        // timeout exceeded ? 
        IF (CheckTimeout(_timerCmd) = RobotLibraryConstants.OK)
        THEN
          ErrorID     := RobotLibraryEvents.ERR_TIMEOUT_CMD;
          ErrorAddTxt := CONCAT('_stepCmd = ' , DINT_TO_STRING(_stepCmd));
        END_IF
      END_IF
  
  
  05: IF (( NOT ExchangeConfiguration.Busy              ) AND
          (     ExchangeConfiguration.ParameterAccepted ))
      THEN
        // stop execution       
        ExchangeConfiguration.Enable := FALSE;
        // set timeout
        SetTimeout(PT := _timeoutCmd, rTimer := _timerCmd);
        // inc step counter
       _stepCmd := _stepCmd + 1;       
       ELSE
         // check error ? 
         IF (ExchangeConfiguration.Error)
         THEN
           ErrorID     := ExchangeConfiguration.ErrorID;
           ErrorAddTxt := ExchangeConfiguration.ErrorAddTxt;;
         END_IF  
       
         // timeout exceeded ? 
         IF (CheckTimeout(_timerCmd) = RobotLibraryConstants.OK)
         THEN
           ErrorID     := RobotLibraryEvents.ERR_TIMEOUT_CMD;
           ErrorAddTxt := CONCAT('_stepCmd = ' , DINT_TO_STRING(_stepCmd));
         END_IF
       END_IF

       
  06: IF (( NOT ReadRobotData.Busy  ) AND 
          ( NOT ReadRobotData.Error )) 
      THEN
        // start function block
        ReadRobotData.Execute := TRUE;
        // set timeout
        SetTimeout(PT := _timeoutCmd, rTimer := _timerCmd);
        // inc step counter
       _stepCmd := _stepCmd + 1;       
      ELSE
        // check error ? 
        IF (ReadRobotData.Error)
        THEN
          ErrorID     := ReadRobotData.ErrorID;
          ErrorAddTxt := ReadRobotData.ErrorAddTxt;;
        END_IF  
        // timeout exceeded ? 
        IF (CheckTimeout(_timerCmd) = RobotLibraryConstants.OK)
        THEN
          ErrorID     := RobotLibraryEvents.ERR_TIMEOUT_CMD;
          ErrorAddTxt := CONCAT('_stepCmd = ' , DINT_TO_STRING(_stepCmd));
        END_IF
      END_IF
  
  07: IF ( ReadRobotData.Busy ) 
      THEN
        // set timeout
        SetTimeout(PT := _timeoutCmd, rTimer := _timerCmd);
        // inc step counter
       _stepCmd := _stepCmd + 1;       
      ELSE
        // check error ? 
        IF (ReadRobotData.Error)
        THEN
          ErrorID     := ReadRobotData.ErrorID;
          ErrorAddTxt := ReadRobotData.ErrorAddTxt;;
        END_IF  
       
        // timeout exceeded ? 
        IF (CheckTimeout(_timerCmd) = RobotLibraryConstants.OK)
        THEN
          ErrorID     := RobotLibraryEvents.ERR_TIMEOUT_CMD;
          ErrorAddTxt := CONCAT('_stepCmd = ' , DINT_TO_STRING(_stepCmd));
        END_IF
      END_IF
  
  
  08: IF (( NOT ReadRobotData.Busy  ) AND
          (     ReadRobotData.Done  ))
      THEN       
        // start function block
        ReadRobotData.Execute := FALSE;
        // set timeout
        SetTimeout(PT := _timeoutCmd, rTimer := _timerCmd);
        // inc step counter
       _stepCmd := _stepCmd + 1;
       ELSE
         // check error ? 
         IF (ReadRobotData.Error)
         THEN
           ErrorID     := ReadRobotData.ErrorID;
           ErrorAddTxt := ReadRobotData.ErrorAddTxt;;
         END_IF  
       
         // timeout exceeded ? 
         IF (CheckTimeout(_timerCmd) = RobotLibraryConstants.OK)
         THEN
           ErrorID     := RobotLibraryEvents.ERR_TIMEOUT_CMD;
           ErrorAddTxt := CONCAT('_stepCmd = ' , DINT_TO_STRING(_stepCmd));
         END_IF
       END_IF


  09: IF (( NOT ReadMessages.Busy  ) AND 
          ( NOT ReadMessages.Error )) 
      THEN
        // start function block
        ReadMessages.Enable := TRUE;
        // set timeout
        SetTimeout(PT := _timeoutCmd, rTimer := _timerCmd);
        // inc step counter
       _stepCmd := _stepCmd + 1;       
      ELSE
        // check error ? 
        IF (ReadMessages.Error)
        THEN
          ErrorID     := ReadMessages.ErrorID;
          ErrorAddTxt := ReadMessages.ErrorAddTxt;;
        END_IF  
        // timeout exceeded ? 
        IF (CheckTimeout(_timerCmd) = RobotLibraryConstants.OK)
        THEN
          ErrorID     := RobotLibraryEvents.ERR_TIMEOUT_CMD;
          ErrorAddTxt := CONCAT('_stepCmd = ' , DINT_TO_STRING(_stepCmd));
        END_IF
      END_IF
  
  10: IF ( ReadMessages.Busy )
      THEN
        // set timeout
        SetTimeout(PT := _timeoutCmd, rTimer := _timerCmd);
        // inc step counter
       _stepCmd := _stepCmd + 1;       
      ELSE
        // check error ? 
        IF (ReadMessages.Error)
        THEN
          ErrorID     := ReadMessages.ErrorID;
          ErrorAddTxt := ReadMessages.ErrorAddTxt;;
        END_IF  
       
        // timeout exceeded ? 
        IF (CheckTimeout(_timerCmd) = RobotLibraryConstants.OK)
        THEN
          ErrorID     := RobotLibraryEvents.ERR_TIMEOUT_CMD;
          ErrorAddTxt := CONCAT('_stepCmd = ' , DINT_TO_STRING(_stepCmd));
        END_IF
      END_IF
  
  
  11: IF ((     ReadMessages.Enabled ) AND
          ( NOT ReadMessages.Error   ))
      THEN       
        // set timeout
        SetTimeout(PT := _timeoutCmd, rTimer := _timerCmd);
        // inc step counter
       _stepCmd := _stepCmd + 1;
      ELSE
         // check error ? 
         IF (ReadRobotData.Error)
         THEN
           ErrorID     := ReadMessages.ErrorID;
           ErrorAddTxt := ReadMessages.ErrorAddTxt;;
         END_IF  
       
         // timeout exceeded ? 
         IF (CheckTimeout(_timerCmd) = RobotLibraryConstants.OK)
         THEN
           ErrorID     := RobotLibraryEvents.ERR_TIMEOUT_CMD;
           ErrorAddTxt := CONCAT('_stepCmd = ' , DINT_TO_STRING(_stepCmd));
         END_IF
       END_IF

  12:  // Reset busy flag
       Busy := FALSE;
       // set initialized flag
       Initialized := TRUE;
       
       // Wait for task disable
       IF ( NOT Enable)
       THEN
         // reset start of function blocks
         ReadMessages.Enable := FALSE;
         ReadRobotData.Execute := FALSE;
         ExchangeConfiguration.Enable := FALSE;
         // Reset step counter
        _stepCmd := 0;         
         // finished okay
         OnExecRun := RobotLibraryConstants.OK;
       END_IF  

       
ELSE
  // invalid step
  ErrorID     := RobotLibraryEvents.ERR_INVALID_STEP;
  ErrorAddTxt := CONCAT('_stepCmd = ' , DINT_TO_STRING(_stepCmd));
END_CASE


// Reset FB
IF ( OnExecRun <> RobotLibraryConstants.RUNNING)
THEN
 _stepCmd     := 0;
  Busy        := FALSE;
  Error       := FALSE;
  ErrorID     := 0;
  ErrorAddTxt := '';
  WarningID   := 0;
  InfoID      := 0;  
END_IF
END_METHOD

METHOD PRIVATE ParseRecvPayload
VAR_IN_OUT
  /// Robot assignment of function
  AxesGroup    : AxesGroup;
  /// Inputs of PLC for communication from RC
  RobotInData  : ARRAY[0..RobotLibraryParameter.ROBOT_IN_DATA_MAX ] OF BYTE;
END_VAR

VAR
  /// internal index
 _idx             : DINT;
  /// temporary DWORD
 _tmpDword        : DWORD;
  /// length of data block
 _dataBlockLength : UINT;
  /// internal payload length
 _payLoadLen      : DWORD;  
  /// internal payload pointer
 _payLoadPtr      : DWORD;  
  /// sequence counter
 _seqCount        : DINT;
END_VAR
// Reset payload
RecvData.Reset();
// Copy inputs to payload  
SysDepMemCpy( pDest := ADR(RecvData.Payload) , pSrc  := ADR(RobotInData), DataLen := RobotLibraryParameter.TELEGRAM_PAYLOAD_MAX +1);

// check new data to receive ? 
IF ( Telegram.RobToPlc.Sequence[0].Header.SEQ_ACK <> AxesGroup.InternalData.LastACK[0]) {warning 'ToDo: handle 2nd sequence'} 
THEN
  // delete old telegram data 
  SysDepMemSet(pDest := ADR(Telegram.RobToPlc), Value := 0 , DataLen := SIZEOF(Telegram.RobToPlc));
END_IF


ParseRecvPayloadHeader        ( AxesGroup := AxesGroup);
ParseRecvPayloadCyclic        ( AxesGroup := AxesGroup);
ParseRecvPayloadCyclicOptional( AxesGroup := AxesGroup);
ParseRecvPayloadSequence      ( AxesGroup := AxesGroup);
ParseRecvPayloadFooter        ( AxesGroup := AxesGroup);
ParseRecvPayloadLogging       ( AxesGroup := AxesGroup);


AxesGroup.InternalData.LastACK[0] := Telegram.RobToPlc.Sequence[0].Header.SEQ_ACK; 
AxesGroup.InternalData.LastACK[1] := Telegram.RobToPlc.Sequence[1].Header.SEQ_ACK;
END_METHOD

METHOD PRIVATE ParseRecvPayloadCyclic
VAR_IN_OUT
  /// Robot assignment of function
  AxesGroup: AxesGroup;
END_VAR
END_METHOD

METHOD PRIVATE ParseRecvPayloadCyclicOptional
VAR_IN_OUT
  /// Robot assignment of function
  AxesGroup    : AxesGroup;
END_VAR

VAR 
  /// internal index for loops
 _idx : DINT;
END_VAR
// AxesGroup.OptionalCyclic.RobToPlc.SubProgramData {{{
IF ( AxesGroup.CyclicOptional.RobToPlc.SubProgramData.Active )
THEN
  FOR _idx := 0 TO 25 {warning 'Add contant for DataMax'}
  DO
    Telegram.RobToPlc.CyclicOptional.SubProgramData.Data[_idx] := RecvData.GetByte(); 
  END_FOR
END_IF
// }}}
  
// AxesGroup.OptionalCyclic.RobToPlc.CartesianPos {{{
IF ( AxesGroup.CyclicOptional.RobToPlc.CartesianPosition.Active )
THEN
  Telegram.RobToPlc.CyclicOptional.CartesianPosition.X                    := RecvData.GetReal();
  Telegram.RobToPlc.CyclicOptional.CartesianPosition.Y                    := RecvData.GetReal();
  Telegram.RobToPlc.CyclicOptional.CartesianPosition.Z                    := RecvData.GetReal();
  Telegram.RobToPlc.CyclicOptional.CartesianPosition.Rx                   := RecvData.GetReal();
  Telegram.RobToPlc.CyclicOptional.CartesianPosition.Ry                   := RecvData.GetReal();
  Telegram.RobToPlc.CyclicOptional.CartesianPosition.Rz                   := RecvData.GetReal();
  Telegram.RobToPlc.CyclicOptional.CartesianPosition.Config               := RecvData.GetWord();
  Telegram.RobToPlc.CyclicOptional.CartesianPosition.Turns_J2_J1          := RecvData.GetByte();
  Telegram.RobToPlc.CyclicOptional.CartesianPosition.Turns_J4_J3          := RecvData.GetByte();
  Telegram.RobToPlc.CyclicOptional.CartesianPosition.Turns_J6_J5          := RecvData.GetByte();
  Telegram.RobToPlc.CyclicOptional.CartesianPosition.Turns_E1             := RecvData.GetByte();  
  Telegram.RobToPlc.CyclicOptional.CartesianPosition.E1                   := RecvData.GetReal();  
  Telegram.RobToPlc.CyclicOptional.CartesianPosition.ToolNo               := RecvData.GetUsint();
  Telegram.RobToPlc.CyclicOptional.CartesianPosition.FrameNo              := RecvData.GetUsint();
  Telegram.RobToPlc.CyclicOptional.CartesianPosition.CurrentlyUsedToolNo  := RecvData.GetUsint();
  Telegram.RobToPlc.CyclicOptional.CartesianPosition.CurrentlyUsedFrameNo := RecvData.GetUsint();
  Telegram.RobToPlc.CyclicOptional.CartesianPosition.Reserve_1            := RecvData.GetByte();
  Telegram.RobToPlc.CyclicOptional.CartesianPosition.Reserve_2            := RecvData.GetByte();  
END_IF
// }}}

// AxesGroup.OptionalCyclic.RobToPlc.JointPosition {{{
IF ( AxesGroup.CyclicOptional.RobToPlc.JointPosition.Active )
THEN
  Telegram.RobToPlc.CyclicOptional.JointPosition.J1         := RecvData.GetReal();
  Telegram.RobToPlc.CyclicOptional.JointPosition.J2         := RecvData.GetReal();
  Telegram.RobToPlc.CyclicOptional.JointPosition.J3         := RecvData.GetReal();
  Telegram.RobToPlc.CyclicOptional.JointPosition.J4         := RecvData.GetReal();
  Telegram.RobToPlc.CyclicOptional.JointPosition.J5         := RecvData.GetReal();
  Telegram.RobToPlc.CyclicOptional.JointPosition.J6         := RecvData.GetReal();
  Telegram.RobToPlc.CyclicOptional.JointPosition.E1         := RecvData.GetReal();
  Telegram.RobToPlc.CyclicOptional.JointPosition.E1_Reserve := RecvData.GetWord();
END_IF  
// }}}

// AxesGroup.OptionalCyclic.RobToPlc.CartesianForce {{{
IF ( AxesGroup.CyclicOptional.RobToPlc.Force.Active )
THEN
  Telegram.RobToPlc.CyclicOptional.Force.X  := RecvData.GetReal();
  Telegram.RobToPlc.CyclicOptional.Force.Y  := RecvData.GetReal();
  Telegram.RobToPlc.CyclicOptional.Force.Z  := RecvData.GetReal();
  Telegram.RobToPlc.CyclicOptional.Force.Rx := RecvData.GetReal();
  Telegram.RobToPlc.CyclicOptional.Force.Ry := RecvData.GetReal();
  Telegram.RobToPlc.CyclicOptional.Force.Rz := RecvData.GetReal();
END_IF  
// }}}    
  
// AxesGroup.OptionalCyclic.RobToPlc.Current {{{
IF ( AxesGroup.CyclicOptional.RobToPlc.Current.Active )
THEN
  Telegram.RobToPlc.CyclicOptional.Current.J1  := RecvData.GetReal();
  Telegram.RobToPlc.CyclicOptional.Current.J2  := RecvData.GetReal();
  Telegram.RobToPlc.CyclicOptional.Current.J3  := RecvData.GetReal();
  Telegram.RobToPlc.CyclicOptional.Current.J4  := RecvData.GetReal();
  Telegram.RobToPlc.CyclicOptional.Current.J5  := RecvData.GetReal();
  Telegram.RobToPlc.CyclicOptional.Current.J6  := RecvData.GetReal();
END_IF    
  
// AxesGroup.OptionalCyclic.RobToPlc.CartesianPosExt {{{
IF ( AxesGroup.CyclicOptional.RobToPlc.CartesianPositionExt.Active )
THEN
  Telegram.RobToPlc.CyclicOptional.CartesianPositionExt.E2 := RecvData.GetReal();
  Telegram.RobToPlc.CyclicOptional.CartesianPositionExt.E3 := RecvData.GetReal();
  Telegram.RobToPlc.CyclicOptional.CartesianPositionExt.E4 := RecvData.GetReal();
  Telegram.RobToPlc.CyclicOptional.CartesianPositionExt.E5 := RecvData.GetReal();
  Telegram.RobToPlc.CyclicOptional.CartesianPositionExt.E6 := RecvData.GetReal();
END_IF  
// }}}       
  
// AxesGroup.OptionalCyclic.RobToPlc.JointPosition {{{
IF ( AxesGroup.CyclicOptional.RobToPlc.JointPositionExt.Active )
THEN
  Telegram.RobToPlc.CyclicOptional.JointPositionExt.E2 := RecvData.GetReal();
  Telegram.RobToPlc.CyclicOptional.JointPositionExt.E3 := RecvData.GetReal();
  Telegram.RobToPlc.CyclicOptional.JointPositionExt.E4 := RecvData.GetReal();
  Telegram.RobToPlc.CyclicOptional.JointPositionExt.E5 := RecvData.GetReal();
  Telegram.RobToPlc.CyclicOptional.JointPositionExt.E6 := RecvData.GetReal();  
END_IF  
// }}}    
      
// AxesGroup.OptionalCyclic.RobToPlc.CartesianForceExt {{{
IF ( AxesGroup.CyclicOptional.RobToPlc.ForceExt.Active )
THEN
  Telegram.RobToPlc.CyclicOptional.ForceExt.E1  := RecvData.GetReal();
  Telegram.RobToPlc.CyclicOptional.ForceExt.E2  := RecvData.GetReal();
  Telegram.RobToPlc.CyclicOptional.ForceExt.E3  := RecvData.GetReal();
  Telegram.RobToPlc.CyclicOptional.ForceExt.E4  := RecvData.GetReal();
  Telegram.RobToPlc.CyclicOptional.ForceExt.E5  := RecvData.GetReal();
  Telegram.RobToPlc.CyclicOptional.ForceExt.E6  := RecvData.GetReal();
END_IF
// }}}    
  
// AxesGroup.OptionalCyclic.RobToPlc.CurrentExt {{{
IF ( AxesGroup.CyclicOptional.RobToPlc.CurrentExt.Active )
THEN
  Telegram.RobToPlc.CyclicOptional.CurrentExt.E1  := RecvData.GetReal();
  Telegram.RobToPlc.CyclicOptional.CurrentExt.E2  := RecvData.GetReal();
  Telegram.RobToPlc.CyclicOptional.CurrentExt.E3  := RecvData.GetReal();
  Telegram.RobToPlc.CyclicOptional.CurrentExt.E4  := RecvData.GetReal();
  Telegram.RobToPlc.CyclicOptional.CurrentExt.E5  := RecvData.GetReal();
  Telegram.RobToPlc.CyclicOptional.CurrentExt.E6  := RecvData.GetReal();
END_IF
// }}}
END_METHOD

METHOD PRIVATE ParseRecvPayloadFooter
VAR_IN_OUT
  /// Robot assignment of function
  AxesGroup : AxesGroup;
END_VAR

VAR
  /// index of lifesign in footer
  _lifeSignIdxFooter : DINT;
END_VAR
IF (( _parCfg.Com.TelegramLengthRobToPlc    >= 1                                          ) AND 
    ( _parCfg.Com.TelegramLengthRobToPlc -1 <= RobotLibraryParameter.TELEGRAM_PAYLOAD_MAX ))
THEN
  // set index of last byte
 _lifeSignIdxFooter := _parCfg.Com.TelegramLengthRobToPlc -1;
 

  Telegram.RobToPlc.Footer.LifeSign := GetHalfeByteHi(RecvData.Payload[_lifeSignIdxFooter]); 
END_IF
END_METHOD

METHOD PRIVATE ParseRecvPayloadHeader
VAR_IN_OUT
  /// Robot assignment of function
  AxesGroup    : AxesGroup;
END_VAR
// Version
Telegram.RobToPlc.Header.SRCIVersion := ByteToVersion(RecvData.GetByte());
// Connection alive signal
Telegram.RobToPlc.Header.LifeSign    := RecvData.GetHalfeByte2(IncPayloadPtr := TRUE);
// Reserved byte
Telegram.RobToPlc.Header.Reserved       := RecvData.GetByte();
// Initialization and Telegram control state
Telegram.RobToPlc.Header.TelegramState  := RecvData.GetUsint();
// Combination of various RA related states.
Telegram.RobToPlc.Header.StatusRobotArm := RecvData.GetDword();
// Actual override in percentage encoding 
Telegram.RobToPlc.Header.Override       := RecvData.GetUint();
END_METHOD

METHOD PRIVATE ParseRecvPayloadLogging
VAR_IN_OUT
  /// Robot assignment of function
  AxesGroup    : AxesGroup;
END_VAR

VAR
  /// internal sequence index for loops
  _seqIdx : DINT;
  /// internal fragment index for loops
  _fragIdx : DINT;
END_VAR
RETURN;
FOR _seqIdx := 0 TO AxesGroup.InternalData.SequenceCountRecv
DO
  // check new data to receive ? 
  IF ( Telegram.RobToPlc.Sequence[_seqIdx].Header.SEQ_ACK <> AxesGroup.InternalData.LastACK[_seqIdx]) 
  THEN
    // Check sequence payload > 0 ?    
    IF (Telegram.RobToPlc.Sequence[_seqIdx].Header.PayloadLength > 0)
    THEN
      // Create log entry
      CreateLogMessagePara4 ( Timestamp   := SystemTime,
                              MessageType := MessageType.CMD,
                              Severity    := Severity.DEBUG,
                              MessageCode := 0,
                              MessageText := 'RecvData: ACK = {1}, received Sequence [{2}] with PayloadLength = {3}, Lifesign = {4}',
                              Para1       :=  UINT_TO_STRING(Telegram.RobToPlc.Sequence[_seqIdx].Header.SEQ_ACK),
                              Para2       :=  DINT_TO_STRING(_seqIdx),
                              Para3       :=  UINT_TO_STRING(Telegram.RobToPlc.Sequence[_seqIdx].Header.PayloadLength),
                              Para4       :=  BYTE_TO_STRING(Telegram.RobToPlc.Header.LifeSign));
  
      FOR _fragIdx := 0 TO AxesGroup.InternalData.FragmentCountRecv[_seqIdx] 
      DO
        // Check fragment payload > 0 ?    
        IF (Telegram.RobToPlc.Sequence[_seqIdx].Fragment[_fragIdx].Header.PayloadLength > 0)
        THEN
          // Create log entry
          CreateLogMessagePara5 ( Timestamp   := SystemTime,
                                  MessageType := MessageType.CMD,
                                  Severity    := Severity.DEBUG,
                                  MessageCode := 0,
                                  MessageText := 'RecvData: received Fragment [{1}] with PayloadLength = {2}, CmdID <{3}> , CmdState: {4}, Fragment-Action Bits: {5}',
                                  Para1       :=  DINT_TO_STRING(0), {warning 'Add seqIdx'}
                                  Para2       :=  UINT_TO_STRING              (Telegram.RobToPlc.Sequence[_seqIdx].Fragment[_fragIdx].Header.PayloadLength),
                                  Para3       :=  DINT_TO_STRING              (Telegram.RobToPlc.Sequence[_seqIdx].Fragment[_fragIdx].Header.CmdID),
                                  Para4       :=  CMD_MESSAGE_STATE_TO_STRING (Telegram.RobToPlc.Sequence[_seqIdx].Fragment[_fragIdx].Command.Header.State),
                                  Para5       :=    FRAGMENT_ACTION_TO_STRING (Telegram.RobToPlc.Sequence[_seqIdx].Fragment[_fragIdx].Header.FragmentAction));
        END_IF
      END_FOR    
    END_IF
  END_IF
END_FOR
END_METHOD

METHOD PRIVATE ParseRecvPayloadSequence
VAR_IN_OUT
  /// Robot assignment of function
  AxesGroup    : AxesGroup;
END_VAR

VAR
  /// internal index
 _idx             : DINT;
  /// temporary DWORD
 _tmpDword        : DWORD;
  /// length of data block
 _dataBlockLength : UINT;
  /// internal payload length
 _payLoadLen      : DWORD;  
  /// internal payload pointer
 _payLoadPtr      : DWORD;  
  /// sequence counter
 _seqCount        : DINT;
END_VAR


VAR_INST
  /// last received acknowledge
 _lastACK : ARRAY[0..1] OF UDINT;
END_VAR
// Sequence Data
Telegram.RobToPlc.Sequence[0].Header.SEQ_ACK       := RecvData.GetUint();
Telegram.RobToPlc.Sequence[0].Header.PayloadLength := RecvData.GetUint();

// check new data ? 
IF ( Telegram.RobToPlc.Sequence[0].Header.SEQ_ACK <> AxesGroup.InternalData.LastACK[0]) {warning 'ToDo Handle 2nd sequence'} 
THEN

  IF (Telegram.RobToPlc.Sequence[0].Header.PayloadLength > 0)
  THEN
    // Create log entry
    CreateLogMessagePara4 ( Timestamp   := SystemTime,
                            MessageType := MessageType.CMD,
                            Severity    := Severity.DEBUG,
                            MessageCode := 0,
                            MessageText := 'RecvData: ACK = {1}, received Sequence [{2}] with PayloadLength = {3}, Lifesign = {4}',
                            Para1       :=  UINT_TO_STRING(Telegram.RobToPlc.Sequence[0].Header.SEQ_ACK),
                            Para2       :=  DINT_TO_STRING(0), {warning 'Add seqIdx'}
                            Para3       :=  UINT_TO_STRING(Telegram.RobToPlc.Sequence[0].Header.PayloadLength),
                            Para4       :=  BYTE_TO_STRING(Telegram.RobToPlc.Header.LifeSign));
    
    Telegram.RobToPlc.Sequence[0].Fragment[0].Header.CmdID               := RecvData.GetUint();
    Telegram.RobToPlc.Sequence[0].Fragment[0].Header.Reserve             := RecvData.GetByte();
    Telegram.RobToPlc.Sequence[0].Fragment[0].Header.FragmentAction      := RecvData.GetByte();
    Telegram.RobToPlc.Sequence[0].Fragment[0].Header.PayloadPointer      := RecvData.GetUint();
    Telegram.RobToPlc.Sequence[0].Fragment[0].Header.PayloadLength       := RecvData.GetUint();
    
    
    IF (Telegram.RobToPlc.Sequence[0].Fragment[0].Header.PayloadLength > 0)
    THEN
      // Fill Respone payload
      FOR _idx := Telegram.RobToPlc.Sequence[0].Fragment[0].Header.PayloadPointer TO Telegram.RobToPlc.Sequence[0].Fragment[0].Header.PayloadLength
      DO
        Telegram.RobToPlc.Sequence[0].Fragment[0].Command.Payload[_idx] := RecvData.GetByte();
      END_FOR
      
      // Add Response to ACR
      AxesGroup.Acyclic.ActiveCommandRegister.AddRsp(Telegram.RobToPlc.Sequence[0].Fragment[0]);
    
      // Only for debugging
      Telegram.RobToPlc.Sequence[0].Fragment[0].Command.Header.State                 := GetHalfeByteLo(Telegram.RobToPlc.Sequence[0].Fragment[0].Command.Payload[0]);
      Telegram.RobToPlc.Sequence[0].Fragment[0].Command.Header.ParSeq                := GetHalfeByteHi(Telegram.RobToPlc.Sequence[0].Fragment[0].Command.Payload[0]);
      Telegram.RobToPlc.Sequence[0].Fragment[0].Command.Header.AlarmMessageSeverity  :=   BYTE_TO_SINT(Telegram.RobToPlc.Sequence[0].Fragment[0].Command.Payload[1]);
      Telegram.RobToPlc.Sequence[0].Fragment[0].Command.Header.AlarmMessageCode      :=  CombineBytesToUint( HiByte := Telegram.RobToPlc.Sequence[0].Fragment[0].Command.Payload[2],
                                                                                                             LoByte := Telegram.RobToPlc.Sequence[0].Fragment[0].Command.Payload[3]);
      // Create log entry
      CreateLogMessagePara5 ( Timestamp   := SystemTime,
                              MessageType := MessageType.CMD,
                              Severity    := Severity.DEBUG,
                              MessageCode := 0,
                              MessageText := 'RecvData: received Fragment [{1}] with PayloadLength = {2}, CmdID <{3}> , CmdState: {4}, Fragment-Action Bits: {5}',
                              Para1       :=  DINT_TO_STRING(0), {warning 'Add seqIdx'}
                              Para2       :=  UINT_TO_STRING              (Telegram.RobToPlc.Sequence[0].Fragment[0].Header.PayloadLength),
                              Para3       :=  DINT_TO_STRING              (Telegram.RobToPlc.Sequence[0].Fragment[0].Header.CmdID),
                              Para4       :=  CMD_MESSAGE_STATE_TO_STRING (Telegram.RobToPlc.Sequence[0].Fragment[0].Command.Header.State),
                              Para5       :=    FRAGMENT_ACTION_TO_STRING (Telegram.RobToPlc.Sequence[0].Fragment[0].Header.FragmentAction));
                              //Para6       :=  BYTE_TO_STRING(Telegram.RobToPlc.Header.LifeSign)
    END_IF    
  END_IF
END_IF  

IF ( RobotLibraryParameter.TWO_SEQUENCES ) {warning 'ToDo'}
THEN
 _seqCount := _seqCount + 1;
END_IF
END_METHOD

END_FUNCTION_BLOCK

// Library/POUs/Read/MC_ReadRobotData/MC_ReadRobotDataFB
/// Read robot-specific data from the RC
FUNCTION_BLOCK MC_ReadRobotDataFB EXTENDS RobotLibraryBaseExecuteFB
// ------------------------------------------------------------------------- 
//  SRCI Robot Library                                                
// ------------------------------------------------------------------------- 
//                                                                           
//  Object:      ReadRobotDataFB                                       
//  Author:      Thorsten Brach                                                
//  Date:        2024-08-11
//
//  Description:                                              
//   
//                                                                           
//  Copyright: 
//    (C) 2024 Thorsten Brach. All rights reserved                                                                                                                                            
//             Licensed under the LGPL-3.0 license.
//                                                                           
//  Disclaimer:                                                                           
//    This project is provided without any guarantee and can be used for   
//    private and commercial purposes. Any use is at the user’s 
//    own risk and responsibility.
//
// -------------------------------------------------------------------------
VAR_INPUT
  /// internal copy of command parameter 
  ParCmd          : ReadRobotDataParCmd;  
END_VAR

VAR_OUTPUT
  /// Command is transferred and confirmed by the RC
  CommandBuffered : BOOL;
  /// command outputs
  OutCmd          : ReadRobotDataOutCmd;       
END_VAR


VAR
  /// internal copy of command parameter 
 _parCmd             : ReadRobotDataParCmd;
  /// command data to send
 _command            : ReadRobotDataSendData;
  /// response data received
 _response           : ReadRobotDataRecvData;      
END_VAR

SUPER^(AxesGroup := AxesGroup);

METHOD PROTECTED CheckFunctionSupported : BOOL
VAR_IN_OUT
  /// Robot assignment of function
  AxesGroup : AxesGroup; 
END_VAR
CheckFunctionSupported := AxesGroup.InternalData.RCSupportedFunctions.ReadRobotData;

IF ( NOT CheckFunctionSupported )
THEN
  // call base implementation for set error and create log entry
  SUPER^.CheckFunctionSupported(AxesGroup := AxesGroup);
END_IF
END_METHOD

METHOD PROTECTED CheckParameterChanged : BOOL
VAR_IN_OUT
  /// Robot assignment of function
  AxesGroup    : AxesGroup; 
END_VAR
// Check ParCmd Size is > 0, because MemCmp does not work correctly with size = 0
IF (SIZEOF(ParCmd) = 0) 
THEN 
  RETURN;
END_IF

// compare memory 
_parameterChanged := ( SysDepMemCmp(pData1 := ADR(ParCmd), pData2 := ADR(_parCmd), DataLen := SIZEOF(ParCmd)) <> RobotLibraryConstants.OK );

// check parameter valid ?
_parameterValid   := CheckParameterValid( AxesGroup := AxesGroup );

IF ((  _parameterChanged        )  AND 
    (  _parameterValid          )) OR
    (  _parameterUpdateInternal )  
THEN  
  // reset internal flag for send parameter update
 _parameterUpdateInternal := FALSE;
  // update internal copy of parameters 
 _parCmd := ParCmd;
  // inc parameter sequence
 _command.ParSeq := _command.ParSeq + 1;
  // update command data  
  CommandData := CreateCommandPayload(AxesGroup := AxesGroup); // ( Access via reference to rCommandFB in ACR )
  // notify active command register 
  AxesGroup.Acyclic.ActiveCommandRegister.NotifyParameterChanged := _uniqueID;
END_IF
END_METHOD

METHOD INTERNAL CreateCommandPayload : RobotLibrarySendDataFB
VAR_IN_OUT
  /// Robot assignment of function
  AxesGroup : AxesGroup; 
END_VAR
// Table 6-17: Sent CMD payload (PLC to RC) of "ReadRobotData"
// --------------------------
// Header
// --------------------------
// Byte 00 : UINT  - Type HB     
// Byte 01 :       - Type LB    
// Byte 02 : USINT - Reserve | ExecutionMode
// Byte 03 : USINT - ParSeq  | Priority
// --------------------------
// set command parameter 
_command.CmdTyp   :=  CmdType.ReadRobotData;
_command.ExecMode :=  ExecMode;
_command.ParSeq   := _command.ParSeq;
_command.Priority :=  Priority;

// copy command data to header
_cmdHeader := _command;
// call base implementation to copy header to payload buffer
CreateCommandPayload := SUPER^.CreateCommandPayload(AxesGroup := AxesGroup);

// Create logging
CreateCommandPayloadLog(AxesGroup := AxesGroup);
END_METHOD

METHOD INTERNAL CreateCommandPayloadLog
VAR_IN_OUT
  /// Robot assignment of function
  AxesGroup : AxesGroup; 
END_VAR
// Create log entry for Parameter start
CreateLogMessage      ( Timestamp   := AxesGroup.InternalData.SystemTime,
                        MessageType := MessageType.CMD,
                        Severity    := Severity.DEBUG,
                        MessageCode := 0,
                        MessageText := 'Create command payload without additional parameter(s)');
END_METHOD

METHOD FB_init : BOOL
VAR_INPUT
  /// if TRUE, the retain variables are initialized (warm start / cold start)
  bInitRetains : BOOL; 
  /// if TRUE, the instance afterwards gets moved into the copy code (online change)
  bInCopyCode  : BOOL;  
END_VAR
MyType := 'MC_ReadRobotDataFB';
ExecMode := ExecutionMode.PARALLEL;
END_METHOD

METHOD PROTECTED OnCall
VAR_IN_OUT
  /// Robot assignment of function
  AxesGroup : AxesGroup; 
END_VAR
// call base implementation
SUPER^.OnCall(AxesGroup := AxesGroup);

CASE _stepCmd OF
  
  00:  IF ( _execute_R.Q )  
       THEN
         // Check function is supported and parameter are valid ?
         IF (( CheckFunctionSupported( AxesGroup := AxesGroup )) AND
             ( CheckParameterValid   ( AxesGroup := AxesGroup )))
         THEN      
           // set busy flag
           Busy := TRUE;
           // Reset command outputs
           SysDepMemSet(pDest := ADR(OutCmd), Value := 0, DataLen := SIZEOF(OutCmd));         
           // apply command parameter
          _parCmd := ParCmd;
           // init parameter sequence
          _command.ParSeq := 1;
           // create command data
           CommandData := CreateCommandPayload(AxesGroup := AxesGroup);
           // Add command to active command register
          _uniqueID := AxesGroup.Acyclic.ActiveCommandRegister.AddCmd( pCommandFB := ADR(THIS^ ));     
           // set timeout
           SetTimeout(PT := _timeoutCmd, rTimer := _timerCmd);
           // inc step counter
          _stepCmd := _stepCmd + 1; 
         END_IF
       END_IF
     

  01:  // Wait for responce received
       IF ( _responseReceived )
       THEN
         // reset response received flag
        _responseReceived := FALSE;

         CASE  _response.State 
         OF
           CmdMessageState.BUFFERED    : CommandBuffered    := TRUE;
           CmdMessageState.DONE        : Done               := TRUE;
           CmdMessageState.ERROR       : Error              := TRUE;
         END_CASE
                
         // Done, Aborted or Error ?
         IF (_response.State >= CmdMessageState.DONE )
         THEN
           // reset Busy Flag
           Busy := FALSE;
           // Update results
           OutCmd.RCManufacturer       :=                              _response.RCManufacturer;
           OutCmd.RCOrderID            :=                              _response.RCOrderID;
           OutCmd.RCSerialNumber       :=                              _response.RCSerialNumber;
           OutCmd.RASerialNumber       :=                              _response.RASerialNumber;
           OutCmd.RCFirmwareVersion    :=                              _response.RCFirmwareVersion;
           OutCmd.RCInterpreterVersion :=                              _response.RCInterpreterVersion;
           OutCmd.AxisJointUsed        :=                              _response.AxisJointUsed;
           OutCmd.AxisExternalUsed     :=                              _response.AxisExternalUsed;
           OutCmd.AxisJointUnit        :=                              _response.AxisJointUnit;
           OutCmd.AxisExternalUnit     :=                              _response.AxisExternalUnit;
           OutCmd.RCSupportedFunctions :=  BytesToRCSupportedFunctions(_response.RCSupportedFunctions);
           OutCmd.RobotID              :=                              _response.RobotID;  
           OutCmd.InterpreterCycleTime :=                              _response.InterpreterCycleTime;
           // set timeout
           SetTimeout(PT := _timeoutCmd, rTimer := _timerCmd);
           // inc step counter
          _stepCmd := _stepCmd + 1; 
         END_IF
       END_IF


  02: IF ( NOT Execute)
      THEN
        Reset();
      END_IF     

ELSE
  // invalid step
  ErrorID := RobotLibraryEvents.ERR_INVALID_STEP;
END_CASE


// Reset FB
IF ( NOT Execute )
THEN
  Reset(); 
END_IF
END_METHOD

METHOD INTERNAL ParseResponsePayload : DINT
VAR_INPUT
  /// Response data
  ResponseData : RobotLibraryRecvDataFB;
  /// Timestamp
  Timestamp    : SystemTime;  
END_VAR
// Table 6-18: Received CMD payload (RC to PLC) of "ReadRobotData"
// --------------------------
// Header
// --------------------------
// Byte 00 : USINT   - ParSeq | State     
// Byte 01 : SINT    - AlarmMessageSeverity    
// Byte 02 : UINT    - AlarmMessageCode HB
// Byte 03 :         - AlarmMessageCode LB
// --------------------------
// Datablock
// --------------------------
// Byte 04 : CHAR  RCManufacturer[0];
// Byte 05 : CHAR  RCManufacturer[1];
// Byte 06 : CHAR  RCManufacturer[2];
// Byte 07 : CHAR  RCManufacturer[3];
// Byte 08 : CHAR  RCManufacturer[4];
// Byte 09 : CHAR  RCManufacturer[5];
// Byte 10 : CHAR  RCManufacturer[6];
// Byte 11 : CHAR  RCManufacturer[7];
// Byte 12 : CHAR  RCManufacturer[8];
// Byte 13 : CHAR  RCManufacturer[9];
// Byte 14 : CHAR  RCManufacturer[10];
// Byte 15 : CHAR  RCManufacturer[11];
// Byte 16 : CHAR  RCManufacturer[12];
// Byte 17 : CHAR  RCManufacturer[13];
// Byte 18 : CHAR  RCManufacturer[14];
// Byte 19 : CHAR  RCManufacturer[15];
// Byte 20 : CHAR  RCManufacturer[16];
// Byte 21 : CHAR  RCManufacturer[17];
// Byte 22 : CHAR  RCManufacturer[18];
// Byte 23 : CHAR  RCManufacturer[19];
// Byte 24 : CHAR  RCOrderID[0];
// Byte 25 : CHAR  RCOrderID[1];
// Byte 26 : CHAR  RCOrderID[2];
// Byte 27 : CHAR  RCOrderID[3];
// Byte 28 : CHAR  RCOrderID[4];
// Byte 29 : CHAR  RCOrderID[5];
// Byte 30 : CHAR  RCOrderID[6];
// Byte 31 : CHAR  RCOrderID[7];
// Byte 32 : CHAR  RCOrderID[8];
// Byte 33 : CHAR  RCOrderID[9];
// Byte 34 : CHAR  RCOrderID[10];
// Byte 35 : CHAR  RCOrderID[11];
// Byte 36 : CHAR  RCOrderID[12];
// Byte 37 : CHAR  RCOrderID[13];
// Byte 38 : CHAR  RCOrderID[14];
// Byte 39 : CHAR  RCOrderID[15];
// Byte 40 : CHAR  RCOrderID[16];
// Byte 41 : CHAR  RCOrderID[17];
// Byte 42 : CHAR  RCOrderID[18];
// Byte 43 : CHAR  RCOrderID[19];
// Byte 44 : CHAR  RCSerialNumber[0];
// Byte 45 : CHAR  RCSerialNumber[1];
// Byte 46 : CHAR  RCSerialNumber[2];
// Byte 47 : CHAR  RCSerialNumber[3];
// Byte 48 : CHAR  RCSerialNumber[4];
// Byte 49 : CHAR  RCSerialNumber[5];
// Byte 50 : CHAR  RCSerialNumber[6];
// Byte 51 : CHAR  RCSerialNumber[7];
// Byte 52 : CHAR  RCSerialNumber[8];
// Byte 53 : CHAR  RCSerialNumber[9];
// Byte 54 : CHAR  RCSerialNumber[10];
// Byte 55 : CHAR  RCSerialNumber[11];
// Byte 56 : CHAR  RCSerialNumber[12];
// Byte 57 : CHAR  RCSerialNumber[13];
// Byte 58 : CHAR  RCSerialNumber[14];
// Byte 59 : CHAR  RCSerialNumber[15];
// Byte 60 : CHAR  RASerialNumber[0];
// Byte 61 : CHAR  RASerialNumber[1];
// Byte 62 : CHAR  RASerialNumber[2];
// Byte 63 : CHAR  RASerialNumber[3];
// Byte 64 : CHAR  RASerialNumber[4];
// Byte 65 : CHAR  RASerialNumber[5];
// Byte 66 : CHAR  RASerialNumber[6];
// Byte 67 : CHAR  RASerialNumber[7];
// Byte 68 : CHAR  RASerialNumber[8];
// Byte 69 : CHAR  RASerialNumber[9];
// Byte 70 : CHAR  RASerialNumber[10];
// Byte 71 : CHAR  RASerialNumber[11];
// Byte 72 : CHAR  RASerialNumber[12];
// Byte 73 : CHAR  RASerialNumber[13];
// Byte 74 : CHAR  RASerialNumber[14];
// Byte 75 : CHAR  RASerialNumber[15];
// Byte 76 : CHAR  RCFirmwareVersion[0];
// Byte 77 : CHAR  RCFirmwareVersion[1];
// Byte 78 : CHAR  RCFirmwareVersion[2];
// Byte 79 : CHAR  RCFirmwareVersion[3];
// Byte 80 : CHAR  RCFirmwareVersion[4];
// Byte 81 : CHAR  RCFirmwareVersion[5];
// Byte 82 : CHAR  RCFirmwareVersion[6];
// Byte 83 : CHAR  RCFirmwareVersion[7];
// Byte 84 : CHAR  RCFirmwareVersion[8];
// Byte 85 : CHAR  RCFirmwareVersion[9];
// Byte 86 : CHAR  RCFirmwareVersion[10];
// Byte 87 : CHAR  RCFirmwareVersion[11];
// Byte 88 : CHAR  RCInterpreterVersion[0];
// Byte 89 : CHAR  RCInterpreterVersion[1];
// Byte 90 : CHAR  RCInterpreterVersion[2];
// Byte 91 : BYTE  Reserved;
// Byte 92 : BYTE  AxisJointUsed;
// Byte 93 : BYTE  AxisExternalUsed;
// Byte 94 : BYTE  AxisJointUnit;
// Byte 95 : BYTE  AxisExternalUnit;
// Byte 96 : BYTE  RCSupportedFunctions[0];
// Byte 97 : BYTE  RCSupportedFunctions[1];
// Byte 98 : BYTE  RCSupportedFunctions[2];
// Byte 99 : BYTE  RCSupportedFunctions[3];
// Byte 100: BYTE  RCSupportedFunctions[4];
// Byte 101: BYTE  RCSupportedFunctions[5];
// Byte 102: BYTE  RCSupportedFunctions[6];
// Byte 103: BYTE  RCSupportedFunctions[7];
// Byte 104: BYTE  RCSupportedFunctions[8];
// Byte 105: BYTE  RCSupportedFunctions[9];
// Byte 106: BYTE  RCSupportedFunctions[10];
// Byte 107: BYTE  RCSupportedFunctions[11];
// Byte 108: BYTE  RCSupportedFunctions[12];
// Byte 109: BYTE  RCSupportedFunctions[13];
// Byte 110: BYTE  RCSupportedFunctions[14];
// Byte 111: BYTE  RCSupportedFunctions[15];
// Byte 112: BYTE  RCSupportedFunctions[16];
// Byte 113: BYTE  RCSupportedFunctions[17];
// Byte 114: BYTE  RCSupportedFunctions[18];
// Byte 115: BYTE  Reserved;
// Byte 116: CHAR  RobotID[0];
// Byte 117: CHAR  RobotID[1];
// Byte 118: CHAR  RobotID[2];
// Byte 119: CHAR  RobotID[3];
// Byte 120: CHAR  RobotID[4];
// Byte 121: CHAR  RobotID[5];
// Byte 122: CHAR  RobotID[6];
// Byte 123: CHAR  RobotID[7];
// Byte 124: CHAR  RobotID[8];
// Byte 125: CHAR  RobotID[9];
// Byte 126: CHAR  RobotID[10];
// Byte 127: CHAR  RobotID[11];
// Byte 128: CHAR  RobotID[12];
// Byte 129: CHAR  RobotID[13];
// Byte 130: CHAR  RobotID[14];
// Byte 131: CHAR  RobotID[15];
// Byte 132: UINT  InterpreterCycleTime HW HB;
// Byte 133:       InterpreterCycleTime HW LB;
// --------------------------
// call base implementation to parse the header from payload buffer
ResponseData.PayloadPtr := SUPER^.ParseResponsePayload(ResponseData := ResponseData, Timestamp := Timestamp);

// copy parsed header to response
_response.ParSeq               := _rspHeader.ParSeq;
_response.State                := _rspHeader.State;
_response.AlarmMessageSeverity := _rspHeader.AlarmMessageSeverity;
_response.AlarmMessageCode     := _rspHeader.AlarmMessageCode;

// Get _response.RCManufacturer
ResponseData.GetDataBlock(pData := ADR(_response.RCManufacturer)      , SIZEOF(_response.RCManufacturer   )   , IsString := TRUE );
// Get _response.RCOrderID
ResponseData.GetDataBlock(pData := ADR(_response.RCOrderID)           , SIZEOF(_response.RCOrderID        )   , IsString := TRUE );
// Get _response.RCSerialNumber
ResponseData.GetDataBlock(pData := ADR(_response.RCSerialNumber)      , SIZEOF(_response.RCSerialNumber   )   , IsString := TRUE );
// Get _response.RASerialNumber
ResponseData.GetDataBlock(pData := ADR(_response.RASerialNumber)      , SIZEOF(_response.RASerialNumber   )   , IsString := TRUE );
// Get _response.RCFirmwareVersion
ResponseData.GetDataBlock(pData := ADR(_response.RCFirmwareVersion)   , SIZEOF(_response.RCFirmwareVersion)   , IsString := TRUE );
// Get _response.RCInterpreterVersion
ResponseData.GetDataBlock(pData := ADR(_response.RCInterpreterVersion), SIZEOF(_response.RCInterpreterVersion), IsString := TRUE );

// Get _response.Reserve
_response.Reserve := ResponseData.GetByte(); 
// Get _response.AxisJointUsed
_response.AxisJointUsed := ResponseData.GetByte(); 
// Get _response.AxisExternalUsed
_response.AxisExternalUsed := ResponseData.GetByte(); 
// Get _response.AxisJointUnit
_response.AxisJointUnit := ResponseData.GetByte(); 
// Get _response.AxisExternalUnit
_response.AxisExternalUnit := ResponseData.GetByte();
// Get _response.RCSupportedFunctions
ResponseData.GetDataBlock(pData := ADR(_response.RCSupportedFunctions), SIZEOF(_response.RCSupportedFunctions), IsString := FALSE );
// Get _response.Reserve2
_response.Reserve2 := ResponseData.GetByte(); 
// Get _response.RobotID
ResponseData.GetDataBlock(pData := ADR(_response.RobotID)             , SIZEOF(_response.RobotID)             , IsString := TRUE );
// Get _response.InterpreterCycleTime
_response.InterpreterCycleTime := ResponseData.GetUsint(); 

// Create logging
ParseResponsePayloadLog(ResponseData := ResponseData, Timestamp := Timestamp);
END_METHOD

METHOD INTERNAL ParseResponsePayloadLog
VAR_INPUT
  /// Response data
  ResponseData : RobotLibraryRecvDataFB;
  /// Timestamp
  Timestamp    : SystemTime;  
END_VAR
VAR 
  /// internal index for loops
 _idx : DINT;
  /// temporary string
 _tmpStr : STRING;
END_VAR
// Create log entry for Parameter start
CreateLogMessage      ( Timestamp   := Timestamp,
                        MessageType := MessageType.CMD,
                        Severity    := Severity.DEBUG,
                        MessageCode := 0,
                        MessageText := 'Parsed the following parameter(s) from response data:');

// Create log entry for RCManufacturer
CreateLogMessagePara1 ( Timestamp   := Timestamp,
                        MessageType := MessageType.CMD,
                        Severity    := Severity.DEBUG,
                        MessageCode := 0,
                        MessageText := 'Response.RCManufacturer = {1}',
                        Para1       := _response.RCManufacturer);

// Create log entry for RCOrderID
CreateLogMessagePara1 ( Timestamp   := Timestamp,
                        MessageType := MessageType.CMD,
                        Severity    := Severity.DEBUG,
                        MessageCode := 0,
                        MessageText := 'Response.RCOrderID = {1}',
                        Para1       := _response.RCOrderID);

// Create log entry for RCSerialNumber
CreateLogMessagePara1 ( Timestamp   := Timestamp,
                        MessageType := MessageType.CMD,
                        Severity    := Severity.DEBUG,
                        MessageCode := 0,
                        MessageText := 'Response.RCSerialNumber = {1}',
                        Para1       := _response.RCSerialNumber);

// Create log entry for RASerialNumber
CreateLogMessagePara1 ( Timestamp   := Timestamp,
                        MessageType := MessageType.CMD,
                        Severity    := Severity.DEBUG,
                        MessageCode := 0,
                        MessageText := 'Response.RASerialNumber = {1}',
                        Para1       := _response.RASerialNumber);

// Create log entry for RCFirmwareVersion
CreateLogMessagePara1 ( Timestamp   := Timestamp,
                        MessageType := MessageType.CMD,
                        Severity    := Severity.DEBUG,
                        MessageCode := 0,
                        MessageText := 'Response.RCFirmwareVersion = {1}',
                        Para1       := _response.RCFirmwareVersion);
                        
// Create log entry for RCInterpreterVersion
CreateLogMessagePara1 ( Timestamp   := Timestamp,
                        MessageType := MessageType.CMD,
                        Severity    := Severity.DEBUG,
                        MessageCode := 0,
                        MessageText := 'Response.RCInterpreterVersion = {1}',
                        Para1       := _response.RCInterpreterVersion);

// Create log entry for Reserve
CreateLogMessagePara1 ( Timestamp   := Timestamp,
                        MessageType := MessageType.CMD,
                        Severity    := Severity.DEBUG,
                        MessageCode := 0,
                        MessageText := 'Response.Reserve = {1}',
                        Para1       :=  BYTE_TO_STRING(_response.Reserve));

// Create log entry for AxisJointUsed
CreateLogMessagePara1 ( Timestamp   := Timestamp,
                        MessageType := MessageType.CMD,
                        Severity    := Severity.DEBUG,
                        MessageCode := 0,
                        MessageText := 'Response.AxisJointUsed = {1}',
                        Para1       :=  BYTE_TO_STRING_BIN(_response.AxisJointUsed));

// Create log entry for AxisExternalUsed
CreateLogMessagePara1 ( Timestamp   := Timestamp,
                        MessageType := MessageType.CMD,
                        Severity    := Severity.DEBUG,
                        MessageCode := 0,
                        MessageText := 'Response.AxisExternalUsed = {1}',
                        Para1       :=  BYTE_TO_STRING_BIN(_response.AxisExternalUsed));

// Create log entry for AxisJointUnit
CreateLogMessagePara1 ( Timestamp   := Timestamp,
                        MessageType := MessageType.CMD,
                        Severity    := Severity.DEBUG,
                        MessageCode := 0,
                        MessageText := 'Response.AxisJointUnit = {1}',
                        Para1       :=  BYTE_TO_STRING(_response.AxisJointUnit));

// Create log entry for AxisExternalUnit
CreateLogMessagePara1 ( Timestamp   := Timestamp,
                        MessageType := MessageType.CMD,
                        Severity    := Severity.DEBUG,
                        MessageCode := 0,
                        MessageText := 'Response.AxisExternalUnit = {1}',
                        Para1       :=  BYTE_TO_STRING(_response.AxisExternalUnit));

FOR _idx := 0 TO 18
do
 _tmpStr := '16#';
 _tmpStr := CONCAT( _tmpStr, BYTE_TO_STRING_BIN(_response.RCSupportedFunctions[_idx]));

  // Create log entry for RCSupportedFunctions
  CreateLogMessagePara2 ( Timestamp   := Timestamp,
                          MessageType := MessageType.CMD,
                          Severity    := Severity.DEBUG,
                          MessageCode := 0,
                          MessageText := 'Response.RCSupportedFunctions[{2}] = {1}',
                          Para1       := _tmpStr,
                          Para2       :=  DINT_TO_STRING(_idx));
END_FOR

// Create log entry for Reserve2
CreateLogMessagePara1 ( Timestamp   := Timestamp,
                        MessageType := MessageType.CMD,
                        Severity    := Severity.DEBUG,
                        MessageCode := 0,
                        MessageText := 'Response.Reserve2 = {1}',
                        Para1       :=  BYTE_TO_STRING(_response.Reserve2));

// Create log entry for RobotID
CreateLogMessagePara1 ( Timestamp   := Timestamp,
                        MessageType := MessageType.CMD,
                        Severity    := Severity.DEBUG,
                        MessageCode := 0,
                        MessageText := 'Response.RobotID = {1}',
                        Para1       :=  _response.RobotID);

// Create log entry for InterpreterCycleTime
CreateLogMessagePara1 ( Timestamp   := Timestamp,
                        MessageType := MessageType.CMD,
                        Severity    := Severity.DEBUG,
                        MessageCode := 0,
                        MessageText := 'Response.InterpreterCycleTime = {1}',
                        Para1       :=  UINT_TO_STRING(_response.InterpreterCycleTime));
END_METHOD

METHOD PROTECTED Reset : DINT
VAR_INPUT
END_VAR
Reset := SUPER^.Reset();

Done               := FALSE;
Busy               := FALSE;
CommandBuffered    := FALSE;
END_METHOD

END_FUNCTION_BLOCK

// Library/POUs/Read/MC_ReadMessages/MC_ReadMessagesFB
/// Read error codes of pending errors and move them into user data block "RobotData"
FUNCTION_BLOCK MC_ReadMessagesFB EXTENDS RobotLibraryBaseEnableFB
// ------------------------------------------------------------------------- 
//  SRCI Robot Library                                                
// ------------------------------------------------------------------------- 
//                                                                           
//  Object:      ReadMessagesFB                                       
//  Author:      Thorsten Brach                                                
//  Date:        2024-06-01
//
//  Description:                                              
//   
//                                                                           
//  Copyright: 
//    (C) 2024 Thorsten Brach. All rights reserved                                                                                                                                            
//             Licensed under the LGPL-3.0 license.
//                                                                           
//  Disclaimer:                                                                           
//    This project is provided without any guarantee and can be used for   
//    private and commercial purposes. Any use is at the user’s 
//    own risk and responsibility.
//
// -------------------------------------------------------------------------
VAR_INPUT
  /// command parameter 
  ParCmd          : ReadMessagesParCmd;
END_VAR
VAR_OUTPUT
  /// TRUE, while the following outputs return valid values:
  /// • Values
  Valid           : BOOL; 
  /// Command is transferred and confirmed by the RC
  CommandBuffered : BOOL;
  /// command outputs
  OutCmd          : ReadMessagesOutCmd;  
END_VAR

VAR
  /// internal copy of command parameter 
 _parCmd             : ReadMessagesParCmd;
  /// command data to send
 _command            : ReadMessagesSendData;
  /// response data received
 _response           : ReadMessagesRecvData;      
END_VAR

SUPER^(AxesGroup := AxesGroup);

METHOD PROTECTED CheckFunctionSupported : BOOL
VAR_IN_OUT
  /// Robot assignment of function
  AxesGroup : AxesGroup; 
END_VAR
CheckFunctionSupported := AxesGroup.InternalData.RCSupportedFunctions.ReadMessages;

IF ( NOT CheckFunctionSupported )
THEN
  // call base implementation for set error and create log entry
  SUPER^.CheckFunctionSupported(AxesGroup := AxesGroup);
END_IF
END_METHOD

METHOD PROTECTED CheckParameterChanged : BOOL
VAR_IN_OUT
  /// Robot assignment of function
  AxesGroup    : AxesGroup; 
END_VAR
// Check ParCmd Size is > 0, because MemCmp does not work correctly with size = 0
IF (SIZEOF(ParCmd) = 0) 
THEN 
  RETURN;
END_IF

// compare memory 
_parameterChanged := ( SysDepMemCmp(pData1 := ADR(ParCmd), pData2 := ADR(_parCmd), DataLen := SIZEOF(ParCmd)) <> RobotLibraryConstants.OK );

// check parameter valid ?
_parameterValid   := CheckParameterValid( AxesGroup := AxesGroup );

IF ((  _parameterChanged        )  AND 
    (  _parameterValid          )) OR
    (  _parameterUpdateInternal )  
THEN  
  // reset internal flag for send parameter update
 _parameterUpdateInternal := FALSE;
  // update internal copy of parameters 
 _parCmd := ParCmd;
  // inc parameter sequence
 _command.ParSeq := _command.ParSeq + 1;
  // update command data  
  CommandData := CreateCommandPayload(AxesGroup := AxesGroup); // ( Access via reference to rCommandFB in ACR )
  // notify active command register 
  AxesGroup.Acyclic.ActiveCommandRegister.NotifyParameterChanged := _uniqueID;
END_IF
END_METHOD

METHOD INTERNAL CreateCommandPayload : RobotLibrarySendDataFB
VAR_IN_OUT
  /// Robot assignment of function
  AxesGroup : AxesGroup; 
END_VAR
// Table 6-107: Sent CMD payload (PLC to RC) of "ReadMessages"
// --------------------------
// Header
// --------------------------
// Byte 00 : UINT  - Type HB     
// Byte 01 :       - Type LB    
// Byte 02 : USINT - Reserve | ExecutionMode
// Byte 03 : USINT - ParSeq  | Priority
// --------------------------
// Datablock
// --------------------------
// Byte 04 : USINT  MsgID;
// Byte 05 : BOOL   Enable;
// Byte 06 : USINT  MessageLevel;
// --------------------------
// set command parameter 
_command.CmdTyp       :=  CmdType.ReadMessages;
_command.ExecMode     :=  ExecMode;
_command.ParSeq       := _command.ParSeq;
_command.Priority     :=  Priority;
_command.MsgID        := _parCmd.MsgID;
_command.Enable       :=  Enable;
_command.MessageLevel := _parCmd.MessageLevel;


// copy command data to header
_cmdHeader := _command;
// call base implementation to copy header to payload buffer
CreateCommandPayload := SUPER^.CreateCommandPayload(AxesGroup := AxesGroup);

// add command.MsgID
CreateCommandPayload.AddUsint(_command.MsgID);
// add command.Enable
CreateCommandPayload.AddBool(_command.Enable);
// add command.MessageLevel
CreateCommandPayload.AddUsint(_command.MessageLevel);

// Create logging
CreateCommandPayloadLog(AxesGroup := AxesGroup);
END_METHOD

METHOD INTERNAL CreateCommandPayloadLog
VAR_IN_OUT
  /// Robot assignment of function
  AxesGroup : AxesGroup; 
END_VAR
// Create log entry for Parameter start
CreateLogMessage      ( Timestamp   := AxesGroup.InternalData.SystemTime,
                        MessageType := MessageType.CMD,
                        Severity    := Severity.DEBUG,
                        MessageCode := 0,
                        MessageText := 'Create command payload with the following parameter(s) :');
  
// Create log entry for MsgID
CreateLogMessagePara1 ( Timestamp   := AxesGroup.InternalData.SystemTime,
                        MessageType := MessageType.CMD,
                        Severity    := Severity.DEBUG,
                        MessageCode := 0,
                        MessageText := 'Command.MsgID = {1}',
                        Para1       :=  USINT_TO_STRING(_command.MsgID));

// Create log entry for Enable
CreateLogMessagePara1 ( Timestamp   := AxesGroup.InternalData.SystemTime,
                        MessageType := MessageType.CMD,
                        Severity    := Severity.DEBUG,
                        MessageCode := 0,
                        MessageText := 'Command.Enable = {1}',
                        Para1       :=  BOOL_TO_STRING(_command.Enable));

// Create log entry for MessageLevel
CreateLogMessagePara1 ( Timestamp   := AxesGroup.InternalData.SystemTime,
                        MessageType := MessageType.CMD,
                        Severity    := Severity.DEBUG,
                        MessageCode := 0,
                        MessageText := 'Command.MessageLevel = {1}',
                        Para1       :=  USINT_TO_STRING(_command.MessageLevel));
END_METHOD

METHOD FB_init : BOOL
VAR_INPUT
  /// if TRUE, the retain variables are initialized (warm start / cold start)
  bInitRetains : BOOL; 
  /// if TRUE, the instance afterwards gets moved into the copy code (online change)
  bInCopyCode  : BOOL;  
END_VAR
MyType := 'MC_ReadMessagesFB';

ExecMode := ExecutionMode.PARALLEL;
END_METHOD

METHOD PROTECTED OnCall
VAR_IN_OUT
  /// Robot assignment of function
  AxesGroup : AxesGroup; 
END_VAR

VAR
  /// internal index for loops
 _idx : DINT;
END_VAR
// call base implementation
SUPER^.OnCall(AxesGroup := AxesGroup);

CASE _stepCmd OF
  
  00:  IF ( _enable_R.Q ) 
       THEN
         // reset the rising edge
        _enable_R();       
         // reset the falling edge
        _enable_F();     
        
         // Check function is supported and parameter are valid ?
         IF (( CheckFunctionSupported( AxesGroup := AxesGroup )) AND
             ( CheckParameterValid   ( AxesGroup := AxesGroup )))
         THEN      
           // set busy flag
           Busy := TRUE;
           // Reset command outputs
           SysDepMemSet(pDest := ADR(OutCmd), Value := 0, DataLen := SIZEOF(OutCmd));         
           // apply command parameter
          _parCmd := ParCmd;
           // init parameter sequence
          _command.ParSeq := 1;
           // create command data
           CommandData := CreateCommandPayload(AxesGroup := AxesGroup);
           // Add command to active command register
          _uniqueID := AxesGroup.Acyclic.ActiveCommandRegister.AddCmd( pCommandFB := ADR(THIS^ ));     
           // set timeout
           SetTimeout(PT := _timeoutCmd, rTimer := _timerCmd);
           // inc step counter
          _stepCmd := _stepCmd + 1;
         END_IF 
       END_IF
     

  01:  // Wait for responce received
       IF ( _responseReceived )
       THEN
         // reset response received flag
        _responseReceived := FALSE;

         CASE  _response.State 
         OF
           CmdMessageState.BUFFERED : CommandBuffered := TRUE;
           CmdMessageState.ERROR    : Error           := TRUE;
           CmdMessageState.ACTIVE   :

           // Update results
           Enabled                       := _response.Enabled OR TRUE; {warning 'ToDo: check why Enabled bit is not set by the RC'}
           OutCmd.MsgId                  := _response.MsgId;
           OutCmd.NumberOfActiveErrors   := _response.NumberOfActiveErrors;
           OutCmd.NumberOfActiveWarnings := _response.NumberOfActiveWarnings;
           OutCmd.Timestamp              := _response.Timestamp;
           OutCmd.MsgType                := _response.MsgType;
           OutCmd.Severity               := _response.Severity;
           OutCmd.ErrorCode              := _response.ErrorCode;
           OutCmd.Text                   := _response.Text;

           // Add message to message buffer           
           AxesGroup.MessageLog.AddMessage(_response);
         END_CASE

         // Done, Aborted or Error ?
         IF (_response.State >= CmdMessageState.DONE )
         THEN
           // Reset Busy flag
           Busy := FALSE;
           // set timeout
           SetTimeout(PT := _timeoutCmd, rTimer := _timerCmd);
           // inc step counter
          _stepCmd := _stepCmd + 1; 
         END_IF
       END_IF

       // do not abort directly, so that the ParSeq update can be send
       IF ( _enable_R.Q ) OR ( _enable_F.Q ) 
       THEN
         // trigger parameter update to disable FB
        _parameterUpdateInternal := TRUE;
         // reset the rising edge
        _enable_R();       
         // reset the falling edge
        _enable_F();       
       END_IF

       
  02: IF (NOT Enable)
      THEN
        Reset();   
      END_IF

ELSE
  // invalid step
  ErrorID := RobotLibraryEvents.ERR_INVALID_STEP;
END_CASE


// Reset FB
IF (( _enable_R.Q ) OR
    ( _enable_F.Q ))
THEN
  Reset();
END_IF
END_METHOD

METHOD INTERNAL ParseResponsePayload : DINT
VAR_INPUT
  /// Response data
  ResponseData : RobotLibraryRecvDataFB;
  /// Timestamp
  Timestamp    : SystemTime;  
END_VAR
// Table 6-108: Received CMD payload (RC to PLC) of "ReadMessages"
// --------------------------
// Header
// --------------------------
// Byte 00 : USINT   - ParSeq | State     
// Byte 01 : SINT    - AlarmMessageSeverity    
// Byte 02 : UINT    - AlarmMessageCode HB
// Byte 03 :         - AlarmMessageCode LB
// --------------------------
// Datablock
// --------------------------
// Byte 04 : BOOL        Enabled;
// Byte 05 : USINT       MsgID;
// Byte 06 : USINT       NumberOfActiveErrors;
// Byte 07 : USINT       NumberOfActiveWarnings;
// Byte 08 : DATE        Date HW HB;
// Byte 09 :             Date HW LB;
// Byte 10 : TIME_OF_DAY Time HW HB;
// Byte 11 :             Time HW LB;
// Byte 12 :             Time LW HB;
// Byte 13 :             Time LW LB;
// Byte 14 : USINT       MsgType;
// Byte 15 : SINT        Severity;
// Byte 16 : DWORD       ErrorCode HW HB;
// Byte 17 :             ErrorCode HW LB;
// Byte 18 :             ErrorCode LW HB;
// Byte 19 :             ErrorCode LW LB;
// Byte 20 : CHAR        Text[0];
// Byte 21 : CHAR        Text[1];
// Byte 22 : CHAR        Text[2];
// Byte 23 : CHAR        Text[3];
// Byte 24 : CHAR        Text[4];
// Byte 25 : CHAR        Text[5];
// Byte 26 : CHAR        Text[6];
// Byte 27 : CHAR        Text[7];
// Byte 28 : CHAR        Text[8];
// Byte 29 : CHAR        Text[9];
// Byte 30 : CHAR        Text[10];
// Byte 31 : CHAR        Text[11];
// Byte 32 : CHAR        Text[12];
// Byte 33 : CHAR        Text[13];
// Byte 34 : CHAR        Text[14];
// Byte 35 : CHAR        Text[15];
// Byte 36 : CHAR        Text[16];
// Byte 37 : CHAR        Text[17];
// Byte 38 : CHAR        Text[18];
// Byte 39 : CHAR        Text[19];
// Byte 40 : CHAR        Text[20];
// Byte 41 : CHAR        Text[21];
// Byte 42 : CHAR        Text[22];
// Byte 43 : CHAR        Text[23];
// Byte 44 : CHAR        Text[24];
// Byte 45 : CHAR        Text[25];
// Byte 46 : CHAR        Text[26];
// Byte 47 : CHAR        Text[27];
// Byte 48 : CHAR        Text[28];
// Byte 49 : CHAR        Text[29];
// Byte 50 : CHAR        Text[30];
// Byte 51 : CHAR        Text[31];
// Byte 52 : CHAR        Text[32];
// Byte 53 : CHAR        Text[33];
// Byte 54 : CHAR        Text[34];
// Byte 55 : CHAR        Text[35];
// Byte 56 : CHAR        Text[36];
// Byte 57 : CHAR        Text[37];
// Byte 58 : CHAR        Text[38];
// Byte 59 : CHAR        Text[39];
// Byte 60 : CHAR        Text[40];
// Byte 61 : CHAR        Text[41];
// Byte 62 : CHAR        Text[42];
// Byte 63 : CHAR        Text[43];
// Byte 64 : CHAR        Text[44];
// Byte 65 : CHAR        Text[45];
// Byte 66 : CHAR        Text[46];
// Byte 67 : CHAR        Text[47];
// Byte 68 : CHAR        Text[48];
// Byte 69 : CHAR        Text[49];
// Byte 70 : CHAR        Text[50];
// Byte 71 : CHAR        Text[51];
// Byte 72 : CHAR        Text[52];
// Byte 73 : CHAR        Text[53];
// Byte 74 : CHAR        Text[54];
// Byte 75 : CHAR        Text[55];
// Byte 76 : CHAR        Text[56];
// Byte 77 : CHAR        Text[57];
// Byte 78 : CHAR        Text[58];
// Byte 79 : CHAR        Text[59];
// Byte 80 : CHAR        Text[60];
// Byte 81 : CHAR        Text[61];
// Byte 82 : CHAR        Text[62];
// Byte 83 : CHAR        Text[63];
// Byte 84 : CHAR        Text[64];
// Byte 85 : CHAR        Text[65];
// Byte 86 : CHAR        Text[66];
// Byte 87 : CHAR        Text[67];
// Byte 88 : CHAR        Text[68];
// Byte 89 : CHAR        Text[69];
// Byte 90 : CHAR        Text[70];
// Byte 91 : CHAR        Text[71];
// Byte 92 : CHAR        Text[72];
// Byte 93 : CHAR        Text[73];
// Byte 94 : CHAR        Text[74];
// Byte 95 : CHAR        Text[75];
// Byte 96 : CHAR        Text[76];
// Byte 97 : CHAR        Text[77];
// Byte 98 : CHAR        Text[78];
// Byte 99 : CHAR        Text[79];
// Byte 100: CHAR        Text[80];
// Byte 101: CHAR        Text[81];
// Byte 102: CHAR        Text[82];
// Byte 103: CHAR        Text[83];
// Byte 104: CHAR        Text[84];
// Byte 105: CHAR        Text[85];
// Byte 106: CHAR        Text[86];
// Byte 107: CHAR        Text[87];
// Byte 108: CHAR        Text[88];
// Byte 109: CHAR        Text[89];
// Byte 110: CHAR        Text[90];
// Byte 111: CHAR        Text[91];
// Byte 112: CHAR        Text[92];
// Byte 113: CHAR        Text[93];
// Byte 114: CHAR        Text[94];
// Byte 115: CHAR        Text[95];
// Byte 116: CHAR        Text[96];
// Byte 117: CHAR        Text[97];
// Byte 118: CHAR        Text[98];
// Byte 119: CHAR        Text[99];
// Byte 120: CHAR        Text[100];
// Byte 121: CHAR        Text[101];
// Byte 122: CHAR        Text[102];
// Byte 123: CHAR        Text[103];
// Byte 124: CHAR        Text[104];
// Byte 125: CHAR        Text[105];
// Byte 126: CHAR        Text[106];
// Byte 127: CHAR        Text[107];
// Byte 128: CHAR        Text[108];
// Byte 129: CHAR        Text[109];
// Byte 130: CHAR        Text[110];
// Byte 131: CHAR        Text[111];
// Byte 132: CHAR        Text[112];
// Byte 133: CHAR        Text[113];
// Byte 134: CHAR        Text[114];
// Byte 135: CHAR        Text[115];
// Byte 136: CHAR        Text[116];
// Byte 137: CHAR        Text[117];
// Byte 138: CHAR        Text[118];
// Byte 139: CHAR        Text[119];
// Byte 140: CHAR        Text[120];
// Byte 141: CHAR        Text[121];
// Byte 142: CHAR        Text[122];
// Byte 143: CHAR        Text[123];
// Byte 144: CHAR        Text[124];
// Byte 145: CHAR        Text[125];
// Byte 146: CHAR        Text[126];
// Byte 147: CHAR        Text[127];
// Byte 148: CHAR        Text[128];
// Byte 149: CHAR        Text[129];
// Byte 150: CHAR        Text[130];
// Byte 151: CHAR        Text[131];
// Byte 152: CHAR        Text[132];
// Byte 153: CHAR        Text[133];
// Byte 154: CHAR        Text[134];
// Byte 155: CHAR        Text[135];
// Byte 156: CHAR        Text[136];
// Byte 157: CHAR        Text[137];
// Byte 158: CHAR        Text[138];
// Byte 159: CHAR        Text[139];
// Byte 160: CHAR        Text[140];
// Byte 161: CHAR        Text[141];
// Byte 162: CHAR        Text[142];
// Byte 163: CHAR        Text[143];
// Byte 164: CHAR        Text[144];
// Byte 165: CHAR        Text[145];
// Byte 166: CHAR        Text[146];
// Byte 167: CHAR        Text[147];
// Byte 168: CHAR        Text[148];
// Byte 169: CHAR        Text[149];
// --------------------------
// call base implementation to parse the header from payload buffer
ResponseData.PayloadPtr := SUPER^.ParseResponsePayload(ResponseData := ResponseData, Timestamp := Timestamp);

// copy parsed header to response
_response.ParSeq               := _rspHeader.ParSeq;
_response.State                := _rspHeader.State;
_response.AlarmMessageSeverity := _rspHeader.AlarmMessageSeverity;
_response.AlarmMessageCode     := _rspHeader.AlarmMessageCode;

// Get Response.Enabled
_response.Enabled := ResponseData.GetBool();
// Get Response.MsgID
_response.MsgID := ResponseData.GetUsint();
// Get Response.NumberOfActiveErrors
_response.NumberOfActiveErrors := ResponseData.GetUsint();
// Get Response.NumberOfActiveWarnings
_response.NumberOfActiveWarnings := ResponseData.GetUsint();
// Get Response.Timestamp.IEC_DATE
_response.Timestamp.IEC_DATE := ResponseData.GetIecDate();
// Get Response.Timestamp.IEC_TIME
_response.Timestamp.IEC_TIME := ResponseData.GetIecTime();
// Get Response.MsgType
_response.MsgType := ResponseData.GetUsint();
// Get Response.Severity
_response.Severity := ResponseData.GetSint();
// Get Response.ErrorCode
_response.ErrorCode := ResponseData.GetDword();
// Get _response.RCManufacturer
ResponseData.GetDataBlock(pData := ADR(_response.Text) , SIZEOF(_response.Text) , IsString := TRUE );

// Create logging
ParseResponsePayloadLog(ResponseData := ResponseData, Timestamp := Timestamp);
END_METHOD

METHOD INTERNAL ParseResponsePayloadLog
VAR_INPUT
  /// Response data
  ResponseData : RobotLibraryRecvDataFB;
  /// Timestamp
  Timestamp    : SystemTime;  
END_VAR
// Create log entry for Parameter start
CreateLogMessage      ( Timestamp   := Timestamp,
                        MessageType := MessageType.CMD,
                        Severity    := Severity.DEBUG,
                        MessageCode := 0,
                        MessageText := 'Parsed the following parameter(s) from response data:');
                        
// Create log entry for Enabled
CreateLogMessagePara1 ( Timestamp   := Timestamp,
                        MessageType := MessageType.CMD,
                        Severity    := Severity.DEBUG,
                        MessageCode := 0,
                        MessageText := 'Response.Enabled = {1}',
                        Para1       :=  BOOL_TO_STRING(_response.Enabled));

// Create log entry for MsgID
CreateLogMessagePara1 ( Timestamp   := Timestamp,
                        MessageType := MessageType.CMD,
                        Severity    := Severity.DEBUG,
                        MessageCode := 0,
                        MessageText := 'Response.MsgID = {1}',
                        Para1       :=  USINT_TO_STRING(_response.MsgID));

// Create log entry for NumberOfActiveErrors
CreateLogMessagePara1 ( Timestamp   := Timestamp,
                        MessageType := MessageType.CMD,
                        Severity    := Severity.DEBUG,
                        MessageCode := 0,
                        MessageText := 'Response.NumberOfActiveErrors = {1}',
                        Para1       :=  USINT_TO_STRING(_response.NumberOfActiveErrors));

// Create log entry for NumberOfActiveWarnings
CreateLogMessagePara1 ( Timestamp   := Timestamp,
                        MessageType := MessageType.CMD,
                        Severity    := Severity.DEBUG,
                        MessageCode := 0,
                        MessageText := 'Response.NumberOfActiveWarnings = {1}',
                        Para1       :=  USINT_TO_STRING(_response.NumberOfActiveWarnings));

// Create log entry for Timestamp.IEC_DATE
CreateLogMessagePara1 ( Timestamp   := Timestamp,
                        MessageType := MessageType.CMD,
                        Severity    := Severity.DEBUG,
                        MessageCode := 0,
                        MessageText := 'Response.Timestamp.IEC_DATE = {1}',
                        Para1       :=  IEC_DATE_TO_STRING(_response.Timestamp.IEC_DATE));

// Create log entry for Timestamp.IEC_TIME
CreateLogMessagePara1 ( Timestamp   := Timestamp,
                        MessageType := MessageType.CMD,
                        Severity    := Severity.DEBUG,
                        MessageCode := 0,
                        MessageText := 'Response.Timestamp.IEC_TIME = {1}',
                        Para1       :=  IEC_TIME_TO_STRING(_response.Timestamp.IEC_TIME));

// Create log entry for MsgType
CreateLogMessagePara1 ( Timestamp   := Timestamp,
                        MessageType := MessageType.CMD,
                        Severity    := Severity.DEBUG,
                        MessageCode := 0,
                        MessageText := 'Response.MsgType = {1}',
                        Para1       :=  USINT_TO_STRING(_response.MsgType));

// Create log entry for Severity
CreateLogMessagePara1 ( Timestamp   := Timestamp,
                        MessageType := MessageType.CMD,
                        Severity    := Severity.DEBUG,
                        MessageCode := 0,
                        MessageText := 'Response.Severity = {1}',
                        Para1       :=  SEVERITY_TO_STRING(_response.Severity,AlignString := FALSE));

// Create log entry for ErrorCode
CreateLogMessagePara1 ( Timestamp   := Timestamp,
                        MessageType := MessageType.CMD,
                        Severity    := Severity.DEBUG,
                        MessageCode := 0,
                        MessageText := 'Response.ErrorCode = {1}',
                        Para1       :=  DWORD_TO_STRING(_response.ErrorCode));

// Create log entry for Text
CreateLogMessagePara1 ( Timestamp   := Timestamp,
                        MessageType := MessageType.CMD,
                        Severity    := Severity.DEBUG,
                        MessageCode := 0,
                        MessageText := 'Response.Text = {1}',
                        Para1       :=  _response.Text);
END_METHOD

METHOD PROTECTED Reset : DINT
VAR_INPUT
END_VAR
Reset := SUPER^.Reset();

Busy               := FALSE;
Valid              := FALSE; 
CommandBuffered    := FALSE;
END_METHOD

END_FUNCTION_BLOCK

// Library/POUs/General/MC_SetOperationMode/MC_SetOperationModeFB
/// Switch operation mode of RC (Automatic External, T1 External, T2 External)
FUNCTION_BLOCK MC_SetOperationModeFB EXTENDS RobotLibraryBaseExecuteFB
// ------------------------------------------------------------------------- 
//  SRCI Robot Library                                                
// ------------------------------------------------------------------------- 
//                                                                           
//  Object:      SetOperationModeFB                                       
//  Author:      Thorsten Brach                                                
//  Date:        2024-06-01
//
//  Description:                                              
//   
//                                                                           
//  Copyright: 
//    (C) 2024 Thorsten Brach. All rights reserved                                                                                                                                            
//             Licensed under the LGPL-3.0 license.
//                                                                           
//  Disclaimer:                                                                           
//    This project is provided without any guarantee and can be used for   
//    private and commercial purposes. Any use is at the user’s 
//    own risk and responsibility.
//
// -------------------------------------------------------------------------
VAR_INPUT
  /// command parameter 
  ParCmd          : SetOperationModeParCmd;
END_VAR
VAR_OUTPUT
  /// Command is transferred and confirmed by the RC
  CommandBuffered : BOOL;
  /// command results
  OutCmd          : SetOperationModeOutCmd;     
END_VAR

VAR
  /// internal copy of command parameter 
 _parCmd          : SetOperationModeParCmd;
  /// command data to send
 _command         : SetOperationModeSendData;
  /// response data received
 _response        : SetOperationModeRecvData;      
END_VAR

SUPER^(AxesGroup := AxesGroup);

METHOD PROTECTED CheckFunctionSupported : BOOL
VAR_IN_OUT
  /// Robot assignment of function
  AxesGroup : AxesGroup; 
END_VAR
CheckFunctionSupported := AxesGroup.InternalData.RCSupportedFunctions.SetOperationMode;

IF ( NOT CheckFunctionSupported )
THEN
  // call base implementation for set error and create log entry
  SUPER^.CheckFunctionSupported(AxesGroup := AxesGroup);
END_IF
END_METHOD

METHOD PROTECTED CheckParameterChanged : BOOL
VAR_IN_OUT
  /// Robot assignment of function
  AxesGroup    : AxesGroup; 
END_VAR
// Check ParCmd Size is > 0, because MemCmp does not work correctly with size = 0
IF (SIZEOF(ParCmd) = 0) 
THEN 
  RETURN;
END_IF

// compare memory 
_parameterChanged := ( SysDepMemCmp(pData1 := ADR(ParCmd), pData2 := ADR(_parCmd), DataLen := SIZEOF(ParCmd)) <> RobotLibraryConstants.OK );

// check parameter valid ?
_parameterValid   := CheckParameterValid( AxesGroup := AxesGroup );

IF ((  _parameterChanged        )  AND 
    (  _parameterValid          )) OR
    (  _parameterUpdateInternal )  
THEN  
  // reset internal flag for send parameter update
 _parameterUpdateInternal := FALSE;
  // update internal copy of parameters 
 _parCmd := ParCmd;
  // inc parameter sequence
 _command.ParSeq := _command.ParSeq + 1;
  // update command data  
  CommandData := CreateCommandPayload(AxesGroup := AxesGroup); // ( Access via reference to rCommandFB in ACR )
  // notify active command register 
  AxesGroup.Acyclic.ActiveCommandRegister.NotifyParameterChanged := _uniqueID;
END_IF
END_METHOD

METHOD INTERNAL CreateCommandPayload : RobotLibrarySendDataFB
VAR_IN_OUT
  /// Robot assignment of function
  AxesGroup : AxesGroup; 
END_VAR
// Table 6-193: Sent CMD payload (PLC to RC) of "SetOperationMode"
// --------------------------
// Header
// --------------------------
// Byte 00 : UINT  - Type HB     
// Byte 01 :       - Type LB    
// Byte 02 : USINT - Reserve | ExecutionMode
// Byte 03 : USINT - ParSeq  | Priority
// --------------------------
// Datablock
// --------------------------
 // Byte 04 : UINT  OperationMode;
 // Byte 05 :       OperationMode;
// --------------------------
// set command parameter 
_command.CmdTyp        :=  CmdType.SetOperationMode;
_command.ExecMode      :=  ExecMode;
_command.ParSeq        := _command.ParSeq;
_command.Priority      :=  Priority;
_command.OperationMode := _parCmd.OperationMode;

// copy command data to header
_cmdHeader := _command;
// call base implementation to copy header to payload buffer
CreateCommandPayload := SUPER^.CreateCommandPayload(AxesGroup := AxesGroup);

// add command.OperationMode
CreateCommandPayload.AddUsint(_command.OperationMode);

// Create logging
CreateCommandPayloadLog(AxesGroup := AxesGroup);
END_METHOD

METHOD INTERNAL CreateCommandPayloadLog 
VAR_IN_OUT
  /// Robot assignment of function
  AxesGroup : AxesGroup; 
END_VAR
// Create log entry for Parameter start
CreateLogMessage      ( Timestamp   := AxesGroup.InternalData.SystemTime,
                        MessageType := MessageType.CMD,
                        Severity    := Severity.DEBUG,
                        MessageCode := 0,
                        MessageText := 'Create command payload with the following parameter(s) :');

// Create log entry for OperationMode
CreateLogMessagePara1 ( Timestamp   := AxesGroup.InternalData.SystemTime,
                        MessageType := MessageType.CMD,
                        Severity    := Severity.DEBUG,
                        MessageCode := 0,
                        MessageText := 'Command.OperationMode = {1}',
                        Para1       :=  USINT_TO_STRING(_command.OperationMode));
END_METHOD

METHOD FB_init : BOOL
VAR_INPUT
  /// if TRUE, the retain variables are initialized (warm start / cold start)
  bInitRetains : BOOL; 
  /// if TRUE, the instance afterwards gets moved into the copy code (online change)
  bInCopyCode  : BOOL;  
END_VAR
MyType := 'MC_SetOperationModeFB';

ExecMode := ExecutionMode.PARALLEL;
END_METHOD

METHOD PROTECTED OnCall
VAR_IN_OUT
  /// Robot assignment of function
  AxesGroup : AxesGroup; 
END_VAR
// call base implementation
SUPER^.OnCall(AxesGroup := AxesGroup);

CASE _stepCmd OF
  
  00:  IF ( _execute_R.Q ) 
       THEN
         // Check function is supported and parameter are valid ?
         IF (( CheckFunctionSupported( AxesGroup := AxesGroup )) AND
             ( CheckParameterValid   ( AxesGroup := AxesGroup )))      
         THEN
           // set busy flag
           Busy := TRUE;
           // Reset command outputs
           SysDepMemSet(pDest := ADR(OutCmd), Value := 0, DataLen := SIZEOF(OutCmd));         
           // apply command parameter
          _parCmd := ParCmd;
           // init parameter sequence
          _command.ParSeq := 1;
           // create command data
           CommandData := CreateCommandPayload(AxesGroup := AxesGroup);
           // Add command to active command register
          _uniqueID := AxesGroup.Acyclic.ActiveCommandRegister.AddCmd( pCommandFB := ADR(THIS^ ));     
           // set timeout
           SetTimeout(PT := _timeoutCmd, rTimer := _timerCmd);
           // inc step counter
          _stepCmd := _stepCmd + 1;
         END_IF 
       END_IF
     

  01:  // Wait for responce received
       IF ( _responseReceived )
       THEN
         // reset response received flag
        _responseReceived := FALSE;

         CASE  _response.State 
         OF
           CmdMessageState.BUFFERED : CommandBuffered := TRUE;
           CmdMessageState.DONE     : Done            := TRUE;
           CmdMessageState.ERROR    : Error           := TRUE;
         END_CASE
                
         // Done, Aborted or Error ?
         IF (_response.State >= CmdMessageState.DONE )
         THEN
           // Reset Busy flag
           Busy := FALSE;
           // set timeout
           SetTimeout(PT := _timeoutCmd, rTimer := _timerCmd);
           // inc step counter
          _stepCmd := _stepCmd + 1; 
         END_IF
       END_IF


  02: IF ( NOT Execute)
      THEN
        Reset();  
      END_IF     

ELSE
  // invalid step
  ErrorID := RobotLibraryEvents.ERR_INVALID_STEP;
END_CASE


// Reset FB
IF ( NOT Execute )
THEN
  Reset(); 
END_IF
END_METHOD

METHOD INTERNAL ParseResponsePayload : DINT
VAR_INPUT
  /// Response data
  ResponseData : RobotLibraryRecvDataFB;
  /// Timestamp
  Timestamp    : SystemTime;  
END_VAR
// Table 6-194: Received CMD payload (RC to PLC) of "SetOperationMode"
// --------------------------
// Header
// --------------------------
// Byte 00 : USINT   - ParSeq | State     
// Byte 01 : SINT    - AlarmMessageSeverity    
// Byte 02 : UINT    - AlarmMessageCode HB
// Byte 03 :         - AlarmMessageCode LB
// --------------------------
// call base implementation to parse the header from payload buffer
ResponseData.PayloadPtr := SUPER^.ParseResponsePayload(ResponseData := ResponseData, Timestamp := Timestamp);

// copy parsed header to response
_response.ParSeq               := _rspHeader.ParSeq;
_response.State                := _rspHeader.State;
_response.AlarmMessageSeverity := _rspHeader.AlarmMessageSeverity;
_response.AlarmMessageCode     := _rspHeader.AlarmMessageCode;

// Create logging
ParseResponsePayloadLog(ResponseData := ResponseData, Timestamp := Timestamp);
END_METHOD

METHOD INTERNAL ParseResponsePayloadLog
VAR_INPUT
  /// Response data
  ResponseData : RobotLibraryRecvDataFB;
  /// Timestamp
  Timestamp    : SystemTime;  
END_VAR
// Create log entry for Parameter start
CreateLogMessage      ( Timestamp   := Timestamp,
                        MessageType := MessageType.CMD,
                        Severity    := Severity.DEBUG,
                        MessageCode := 0,
                        MessageText := 'Parsed the following parameter(s) from response data:');
                        
// Create log entry for no parameter 
CreateLogMessage      ( Timestamp   := Timestamp,
                        MessageType := MessageType.CMD,
                        Severity    := Severity.DEBUG,
                        MessageCode := 0,
                        MessageText := 'This command has no parameter to parse...');
END_METHOD

METHOD PROTECTED Reset : DINT
VAR_INPUT
END_VAR
Reset := SUPER^.Reset();

Done               := FALSE;
Busy               := FALSE;
CommandBuffered    := FALSE;
END_METHOD

END_FUNCTION_BLOCK

// Library/POUs/General/MC_SetSequence/MC_SetSequenceFB
/// Set active sequence
FUNCTION_BLOCK MC_SetSequenceFB EXTENDS RobotLibraryBaseExecuteFB
// ------------------------------------------------------------------------- 
//  SRCI Robot Library                                                
// ------------------------------------------------------------------------- 
//                                                                           
//  Object:      SetSequenceFB                                       
//  Author:      Thorsten Brach                                                
//  Date:        2024-06-01
//
//  Description:                                              
//   
//                                                                           
//  Copyright: 
//    (C) 2024 Thorsten Brach. All rights reserved                                                                                                                                            
//             Licensed under the LGPL-3.0 license.
//                                                                           
//  Disclaimer:                                                                           
//    This project is provided without any guarantee and can be used for   
//    private and commercial purposes. Any use is at the user’s 
//    own risk and responsibility.
//
// -------------------------------------------------------------------------
VAR_INPUT
  /// command parameter 
  ParCmd          : SetSequenceParCmd;  
END_VAR

VAR_OUTPUT
  /// Command is transferred and confirmed by the RC
  CommandBuffered : BOOL;
  /// command results
  OutCmd          : SetSequenceOutCmd;     
END_VAR

VAR
  /// internal copy of command parameter 
 _parCmd          : SetSequenceParCmd;
  /// command data to send
 _command         : SetSequenceSendData;
  /// response data received
 _response        : SetSequenceRecvData;      
END_VAR

SUPER^(AxesGroup := AxesGroup);

METHOD PROTECTED CheckFunctionSupported : BOOL
VAR_IN_OUT
  /// Robot assignment of function
  AxesGroup : AxesGroup; 
END_VAR
CheckFunctionSupported := AxesGroup.InternalData.RCSupportedFunctions.SetSequence;

IF ( NOT CheckFunctionSupported )
THEN
  // call base implementation for set error and create log entry
  SUPER^.CheckFunctionSupported(AxesGroup := AxesGroup);
END_IF
END_METHOD

METHOD PROTECTED CheckParameterChanged : BOOL
VAR_IN_OUT
  /// Robot assignment of function
  AxesGroup    : AxesGroup; 
END_VAR
// Check ParCmd Size is > 0, because MemCmp does not work correctly with size = 0
IF (SIZEOF(ParCmd) = 0) 
THEN 
  RETURN;
END_IF

// compare memory 
_parameterChanged := ( SysDepMemCmp(pData1 := ADR(ParCmd), pData2 := ADR(_parCmd), DataLen := SIZEOF(ParCmd)) <> RobotLibraryConstants.OK );

// check parameter valid ?
_parameterValid   := CheckParameterValid( AxesGroup := AxesGroup );

IF ((  _parameterChanged        )  AND 
    (  _parameterValid          )) OR
    (  _parameterUpdateInternal )  
THEN  
  // reset internal flag for send parameter update
 _parameterUpdateInternal := FALSE;
  // update internal copy of parameters 
 _parCmd := ParCmd;
  // inc parameter sequence
 _command.ParSeq := _command.ParSeq + 1;
  // update command data  
  CommandData := CreateCommandPayload(AxesGroup := AxesGroup); // ( Access via reference to rCommandFB in ACR )
  // notify active command register 
  AxesGroup.Acyclic.ActiveCommandRegister.NotifyParameterChanged := _uniqueID;
END_IF
END_METHOD

METHOD INTERNAL CreateCommandPayload : RobotLibrarySendDataFB
VAR_IN_OUT
  /// Robot assignment of function
  AxesGroup : AxesGroup; 
END_VAR
// Table 6-92: Sent CMD payload (PLC to RC) of "SetSequence"
// --------------------------
// Header
// --------------------------
// Byte 00 : UINT  - Type HB     
// Byte 01 :       - Type LB    
// Byte 02 : USINT - Reserve | ExecutionMode
// Byte 03 : USINT - ParSeq  | Priority
// --------------------------
// Datablock
// --------------------------
// Byte 04 : UINT  TargetSequence;
// set command parameter 
_command.CmdTyp         :=  CmdType.SetSequence;
_command.ExecMode       :=  ExecMode;
_command.ParSeq         := _command.ParSeq;
_command.Priority       :=  Priority;
_command.TargetSequence := _parCmd.TargetSequence;

// copy command data to header
_cmdHeader := _command;
// call base implementation to copy header to payload buffer
CreateCommandPayload := SUPER^.CreateCommandPayload(AxesGroup := AxesGroup);

// add command.TargetSequence
CreateCommandPayload.AddUsint(_command.TargetSequence);

// Create logging
CreateCommandPayloadLog(AxesGroup := AxesGroup);
END_METHOD

METHOD INTERNAL CreateCommandPayloadLog 
VAR_IN_OUT
  /// Robot assignment of function
  AxesGroup : AxesGroup; 
END_VAR
// Create log entry for Parameter start
CreateLogMessage      ( Timestamp   := AxesGroup.InternalData.SystemTime,
                        MessageType := MessageType.CMD,
                        Severity    := Severity.DEBUG,
                        MessageCode := 0,
                        MessageText := 'Create command payload with the following parameter(s) :');

// Create log entry for TargetSequence
CreateLogMessagePara1 ( Timestamp   := AxesGroup.InternalData.SystemTime,
                        MessageType := MessageType.CMD,
                        Severity    := Severity.DEBUG,
                        MessageCode := 0,
                        MessageText := 'Command.TargetSequence = {1}',
                        Para1       :=  USINT_TO_STRING(_command.TargetSequence));
END_METHOD

METHOD FB_init : BOOL
VAR_INPUT
  /// if TRUE, the retain variables are initialized (warm start / cold start)
  bInitRetains : BOOL; 
  /// if TRUE, the instance afterwards gets moved into the copy code (online change)
  bInCopyCode  : BOOL;  
END_VAR
MyType := 'MC_SetSequenceFB';

ExecMode := ExecutionMode.PARALLEL;
END_METHOD

METHOD PROTECTED OnCall
VAR_IN_OUT
  /// Robot assignment of function
  AxesGroup : AxesGroup; 
END_VAR
// call base implementation
SUPER^.OnCall(AxesGroup := AxesGroup);

CASE _stepCmd OF
  
  00:  IF ( _execute_R.Q )  
       THEN
         // Check function is supported and parameter are valid ?
         IF (( CheckFunctionSupported( AxesGroup := AxesGroup )) AND
             ( CheckParameterValid   ( AxesGroup := AxesGroup )))      
         THEN
           // set busy flag
           Busy := TRUE;
           // Reset command outputs
           SysDepMemSet(pDest := ADR(OutCmd), Value := 0, DataLen := SIZEOF(OutCmd));         
           // apply command parameter
          _parCmd := ParCmd;
           // init parameter sequence
          _command.ParSeq := 1;
           // create command data
           CommandData := CreateCommandPayload(AxesGroup := AxesGroup);
           // Add command to active command register
          _uniqueID := AxesGroup.Acyclic.ActiveCommandRegister.AddCmd( pCommandFB := ADR(THIS^ ));     
           // set timeout
           SetTimeout(PT := _timeoutCmd, rTimer := _timerCmd);
           // inc step counter
          _stepCmd := _stepCmd + 1;
         END_IF 
       END_IF
     

  01:  // Wait for responce received
       IF ( _responseReceived )
       THEN
         // reset response received flag
        _responseReceived := FALSE;

         CASE  _response.State 
         OF
           CmdMessageState.BUFFERED : CommandBuffered := TRUE;
           CmdMessageState.DONE     : Done            := TRUE;
           CmdMessageState.ERROR    : Error           := TRUE;
         END_CASE
                
         // Done, Aborted or Error ?
         IF (_response.State >= CmdMessageState.DONE )
         THEN
           // Reset Busy flag
           Busy:= FALSE;
           // set timeout
           SetTimeout(PT := _timeoutCmd, rTimer := _timerCmd);
           // inc step counter
          _stepCmd := _stepCmd + 1; 
         END_IF
       END_IF


  02: IF ( NOT Execute)
      THEN
        Reset();
      END_IF     

ELSE
  // invalid step
  ErrorID := RobotLibraryEvents.ERR_INVALID_STEP;
END_CASE


// Reset FB
IF ( NOT Execute )
THEN
  Reset();
END_IF
END_METHOD

METHOD INTERNAL ParseResponsePayload : DINT
VAR_INPUT
  /// Response data
  ResponseData : RobotLibraryRecvDataFB;
  /// Timestamp
  Timestamp    : SystemTime;  
END_VAR
// Table 6-93: Received CMD payload (RC to PLC) of "SetSequence"
// --------------------------
// Header
// --------------------------
// Byte 00 : USINT   - ParSeq | State     
// Byte 01 : SINT    - AlarmMessageSeverity    
// Byte 02 : UINT    - AlarmMessageCode HB
// Byte 03 :         - AlarmMessageCode LB
// call base implementation to parse the header from payload buffer
ResponseData.PayloadPtr := SUPER^.ParseResponsePayload(ResponseData := ResponseData, Timestamp := Timestamp);

// copy parsed header to response
_response.ParSeq               := _rspHeader.ParSeq;
_response.State                := _rspHeader.State;
_response.AlarmMessageSeverity := _rspHeader.AlarmMessageSeverity;
_response.AlarmMessageCode     := _rspHeader.AlarmMessageCode;

// Create logging
ParseResponsePayloadLog(ResponseData := ResponseData, Timestamp := Timestamp);
END_METHOD

METHOD INTERNAL ParseResponsePayloadLog
VAR_INPUT
  /// Response data
  ResponseData : RobotLibraryRecvDataFB;
  /// Timestamp
  Timestamp    : SystemTime;  
END_VAR
// Create log entry for Parameter start
CreateLogMessage      ( Timestamp   := Timestamp,
                        MessageType := MessageType.CMD,
                        Severity    := Severity.DEBUG,
                        MessageCode := 0,
                        MessageText := 'Parsed the following parameter(s) from response data:');
                        
// Create log entry for no parameter 
CreateLogMessage      ( Timestamp   := Timestamp,
                        MessageType := MessageType.CMD,
                        Severity    := Severity.DEBUG,
                        MessageCode := 0,
                        MessageText := 'This command has no parameter to parse...');
END_METHOD

METHOD PROTECTED Reset : DINT
VAR_INPUT
END_VAR
Reset := SUPER^.Reset();

Done               := FALSE;
Busy               := FALSE;
CommandBuffered    := FALSE;
END_METHOD

END_FUNCTION_BLOCK

// Library/POUs/General/MC_SwitchLanguage/MC_SwitchLanguageFB
/// Switch language of robot teach pendant from PLC
FUNCTION_BLOCK MC_SwitchLanguageFB EXTENDS RobotLibraryBaseExecuteFB
// ------------------------------------------------------------------------- 
//  SRCI Robot Library                                                
// ------------------------------------------------------------------------- 
//                                                                           
//  Object:      SwitchLanguageFB                                       
//  Author:      Thorsten Brach                                                
//  Date:        2024-06-01
//
//  Description:                                              
//   
//                                                                           
//  Copyright: 
//    (C) 2024 Thorsten Brach. All rights reserved                                                                                                                                            
//             Licensed under the LGPL-3.0 license.
//                                                                           
//  Disclaimer:                                                                           
//    This project is provided without any guarantee and can be used for   
//    private and commercial purposes. Any use is at the user’s 
//    own risk and responsibility.
//
// -------------------------------------------------------------------------
VAR_INPUT
  /// Command parameter 
  ParCmd          : SwitchLanguageParCmd;    
END_VAR

VAR_OUTPUT
  /// Command is transferred and confirmed by the RC
  CommandBuffered : BOOL;
  /// command results
  OutCmd          : SwitchLanguageOutCmd;     
END_VAR

VAR
  /// internal copy of command parameter 
 _parCmd          : SwitchLanguageParCmd;
  /// command data to send
 _command         : SwitchLanguageSendData;
  /// response data received
 _response        : SwitchLanguageRecvData;      
END_VAR

SUPER^(AxesGroup := AxesGroup);

METHOD PROTECTED CheckFunctionSupported : BOOL
VAR_IN_OUT
  /// Robot assignment of function
  AxesGroup : AxesGroup; 
END_VAR
CheckFunctionSupported := AxesGroup.InternalData.RCSupportedFunctions.SwitchLanguage;

IF ( NOT CheckFunctionSupported )
THEN
  // call base implementation for set error and create log entry
  SUPER^.CheckFunctionSupported(AxesGroup := AxesGroup);
END_IF
END_METHOD

METHOD PROTECTED CheckParameterChanged : BOOL
VAR_IN_OUT
  /// Robot assignment of function
  AxesGroup    : AxesGroup; 
END_VAR
// Check ParCmd Size is > 0, because MemCmp does not work correctly with size = 0
IF (SIZEOF(ParCmd) = 0) 
THEN 
  RETURN;
END_IF

// compare memory 
_parameterChanged := ( SysDepMemCmp(pData1 := ADR(ParCmd), pData2 := ADR(_parCmd), DataLen := SIZEOF(ParCmd)) <> RobotLibraryConstants.OK );

// check parameter valid ?
_parameterValid   := CheckParameterValid( AxesGroup := AxesGroup );

IF ((  _parameterChanged        )  AND 
    (  _parameterValid          )) OR
    (  _parameterUpdateInternal )  
THEN  
  // reset internal flag for send parameter update
 _parameterUpdateInternal := FALSE;
  // update internal copy of parameters 
 _parCmd := ParCmd;
  // inc parameter sequence
 _command.ParSeq := _command.ParSeq + 1;
  // update command data  
  CommandData := CreateCommandPayload(AxesGroup := AxesGroup); // ( Access via reference to rCommandFB in ACR )
  // notify active command register 
  AxesGroup.Acyclic.ActiveCommandRegister.NotifyParameterChanged := _uniqueID;
END_IF
END_METHOD

METHOD INTERNAL CreateCommandPayload : RobotLibrarySendDataFB
VAR_IN_OUT
  /// Robot assignment of function
  AxesGroup : AxesGroup; 
END_VAR
// Table 6-76: Sent CMD payload (PLC to RC) of "SwitchLanguage"
// --------------------------
// Header
// --------------------------
// Byte 00 : UINT  - Type HB     
// Byte 01 :       - Type LB    
// Byte 02 : USINT - Reserve | ExecutionMode
// Byte 03 : USINT - ParSeq  | Priority
// --------------------------
// Datablock
// --------------------------
// Byte 04 : STRING(2)  - LanguageCode[0]
// Byte 05 :            - LanguageCode[1]
// set command parameter 
_command.CmdTyp       :=  CmdType.SwitchLanguage;
_command.ExecMode     :=  ExecMode;
_command.ParSeq       := _command.ParSeq;
_command.Priority     :=  Priority;

_command.LanguageCode := _parCmd.LanguageCode;


// copy command data to header
_cmdHeader := _command;
// call base implementation to copy header to payload buffer
CreateCommandPayload := SUPER^.CreateCommandPayload(AxesGroup := AxesGroup);

// add command.LanguageCode
CreateCommandPayload.AddString(_command.LanguageCode);

// Create logging
CreateCommandPayloadLog(AxesGroup := AxesGroup);
END_METHOD

METHOD INTERNAL CreateCommandPayloadLog 
VAR_IN_OUT
  /// Robot assignment of function
  AxesGroup : AxesGroup; 
END_VAR
// Create log entry for Parameter start
CreateLogMessage      ( Timestamp   := AxesGroup.InternalData.SystemTime,
                        MessageType := MessageType.CMD,
                        Severity    := Severity.DEBUG,
                        MessageCode := 0,
                        MessageText := 'Create command payload with the following parameter(s) :');

// Create log entry for LanguageCode
CreateLogMessagePara1 ( Timestamp   := AxesGroup.InternalData.SystemTime,
                        MessageType := MessageType.CMD,
                        Severity    := Severity.DEBUG,
                        MessageCode := 0,
                        MessageText := 'Command.LanguageCode = {1}',
                        Para1       :=  _command.LanguageCode);
END_METHOD

METHOD FB_init : BOOL
VAR_INPUT
  /// if TRUE, the retain variables are initialized (warm start / cold start)
  bInitRetains : BOOL; 
  /// if TRUE, the instance afterwards gets moved into the copy code (online change)
  bInCopyCode  : BOOL;  
END_VAR
MyType := 'MC_SwitchLanguageFB';

ExecMode := ExecutionMode.PARALLEL;
END_METHOD

METHOD PROTECTED OnCall
VAR_IN_OUT
  /// Robot assignment of function
  AxesGroup : AxesGroup; 
END_VAR
// call base implementation
SUPER^.OnCall(AxesGroup := AxesGroup);

CASE _stepCmd OF
  
  00:  IF ( _execute_R.Q )  
       THEN
         // Check function is supported and parameter are valid ?
         IF (( CheckFunctionSupported( AxesGroup := AxesGroup )) AND
             ( CheckParameterValid   ( AxesGroup := AxesGroup )))      
         THEN
           // set busy flag
           Busy := TRUE;
           // Reset command outputs
           SysDepMemSet(pDest := ADR(OutCmd), Value := 0, DataLen := SIZEOF(OutCmd));         
           // apply command parameter
          _parCmd := ParCmd;
           // init parameter sequence
          _command.ParSeq := 1;
           // create command data
           CommandData := CreateCommandPayload(AxesGroup := AxesGroup);
           // Add command to active command register
          _uniqueID := AxesGroup.Acyclic.ActiveCommandRegister.AddCmd( pCommandFB := ADR(THIS^ ));     
           // set timeout
           SetTimeout(PT := _timeoutCmd, rTimer := _timerCmd);
           // inc step counter
          _stepCmd := _stepCmd + 1;
         END_IF 
       END_IF
     

  01:  // Wait for responce received
       IF ( _responseReceived )
       THEN
         // reset response received flag
        _responseReceived := FALSE;

         CASE  _response.State 
         OF
           CmdMessageState.BUFFERED : CommandBuffered := TRUE;
           CmdMessageState.DONE     : Done            := TRUE;
           CmdMessageState.ERROR    : Error           := TRUE;
         END_CASE
                
         // Done, Aborted or Error ?
         IF (_response.State >= CmdMessageState.DONE )
         THEN
           // Reset Busy flag
           Busy := FALSE;
           // Update results
           OutCmd.ActualLanguageCode := _response.ActualLanguageCode;
           // set timeout
           SetTimeout(PT := _timeoutCmd, rTimer := _timerCmd);
           // inc step counter
          _stepCmd := _stepCmd + 1; 
         END_IF
       END_IF


  02: IF ( NOT Execute)
      THEN
        Reset();
      END_IF     

ELSE
  // invalid step
  ErrorID := RobotLibraryEvents.ERR_INVALID_STEP;
END_CASE


// Reset FB
IF ( NOT Execute )
THEN
  Reset();
END_IF
END_METHOD

